   1:  PR[91,2] = PR[90,2] + -2.008;
   1:  PR[91,3] = PR[90,3] + 3.667;
   1:L PR[91] R[100]mm/sec CNT100;
   1:  PR[91,1] = PR[90,1] + -36.732;
   1:  PR[91,2] = PR[90,2] + -2.668;
   1:  PR[91,3] = PR[90,3] + 3.670;
   1:L PR[91] R[100]mm/sec CNT100;
   1:  PR[91,1] = PR[90,1] + -36.503;
   1:  PR[91,2] = PR[90,2] + -3.709;
   1:  PR[91,3] = PR[90,3] + 3.674;
   1:L PR[91] R[100]mm/sec CNT100;
   1:  PR[91,1] = PR[90,1] + -36.318;
   1:  PR[91,2] = PR[90,2] + -4.391;
   1:  PR[91,3] = PR[90,3] + 3.681;
   1:L PR[91] R[100]mm/sec CNT100;
   1:  PR[91,1] = PR[90,1] + -35.924;
   1:  PR[91,2] = PR[90,2] + -5.558;
   1:  PR[91,3] = PR[90,3] + 3.685;
   1:L PR[91] R[100]mm/sec CNT100;
   1:  PR[91,1] = PR[90,1] + -35.717;
   1:  PR[91,2] = PR[90,2] + -6.077;
   1:  PR[91,3] = PR[90,3] + 3.693;
   1:L PR[91] R[100]mm/sec CNT100;
   1:  PR[91,1] = PR[90,1] + -35.452;
   1:  PR[91,2] = PR[90,2] + -6.678;
   1:  PR[91,3] = PR[90,3] + 3.696;
   1:L PR[91] R[100]mm/sec CNT100;
   1:  PR[91,1] = PR[90,1] + -35.136;
   1:  PR[91,2] = PR[90,2] + -7.322;
   1:  PR[91,3] = PR[90,3] + 3.700;
   1:L PR[91] R[100]mm/sec CNT100;
   1:  PR[91,1] = PR[90,1] + -34.899;
   1:  PR[91,2] = PR[90,2] + -7.767;
   1:  PR[91,3] = PR[90,3] + 3.704;
   1:L PR[91] R[100]mm/sec CNT100;
   1:  PR[91,1] = PR[90,1] + -34.544;
   1:  PR[91,2] = PR[90,2] + -8.374;
   1:  PR[91,3] = PR[90,3] + 3.708;
   1:L PR[91] R[100]mm/sec CNT100;
   1:  PR[91,1] = PR[90,1] + -33.978;
   1:  PR[91,2] = PR[90,2] + -9.242;
   1:  PR[91,3] = PR[90,3] + 3.712;
   1:L PR[91] R[100]mm/sec CNT100;
   1:  PR[91,1] = PR[90,1] + -33.867;
   1:  PR[91,2] = PR[90,2] + -9.398;
   1:  PR[91,3] = PR[90,3] + 3.718;
   1:L PR[91] R[100]mm/sec CNT100;
   1:  PR[91,1] = PR[90,1] + -33.245;
   1:  PR[91,2] = PR[90,2] + -10.215;
   1:  PR[91,3] = PR[90,3] + 3.719;
   1:L PR[91] R[100]mm/sec CNT100;
   1:  PR[91,1] = PR[90,1] + -32.790;
   1:  PR[91,2] = PR[90,2] + -10.756;
   1:  PR[91,3] = PR[90,3] + 3.725;
   1:L PR[91] R[100]mm/sec CNT100;
   1:  PR[91,1] = PR[90,1] + -31.941;
   1:  PR[91,2] = PR[90,2] + -11.649;
   1:  PR[91,3] = PR[90,3] + 3.730;
   1:L PR[91] R[100]mm/sec CNT100;
   1:  PR[91,1] = PR[90,1] + -31.042;
   1:  PR[91,2] = PR[90,2] + -12.468;
   1:  PR[91,3] = PR[90,3] + 3.737;
   1:L PR[91] R[100]mm/sec CNT100;
   1:  PR[91,1] = PR[90,1] + -30.081;
   1:  PR[91,2] = PR[90,2] + -13.224;
   1:  PR[91,3] = PR[90,3] + 3.745;
   1:L PR[91] R[100]mm/sec CNT100;
   1:  PR[91,1] = PR[90,1] + -29.069;
   1:  PR[91,2] = PR[90,2] + -13.908;
   1:  PR[91,3] = PR[90,3] + 3.752;
   1:L PR[91] R[100]mm/sec CNT100;
   1:  PR[91,1] = PR[90,1] + -27.991;
   1:  PR[91,2] = PR[90,2] + -14.526;
   1:  PR[91,3] = PR[90,3] + 3.759;
   1:L PR[91] R[100]mm/sec CNT100;
   1:  PR[91,1] = PR[90,1] + -26.909;
   1:  PR[91,2] = PR[90,2] + -15.048;
   1:  PR[91,3] = PR[90,3] + 3.767;
   1:L PR[91] R[100]mm/sec CNT100;
   1:  PR[91,1] = PR[90,1] + -25.772;
   1:  PR[91,2] = PR[90,2] + -15.498;
   1:  PR[91,3] = PR[90,3] + 3.774;
   1:L PR[91] R[100]mm/sec CNT100;
   1:  PR[91,1] = PR[90,1] + -24.607;
   1:  PR[91,2] = PR[90,2] + -15.865;
   1:  PR[91,3] = PR[90,3] + 3.782;
   1:L PR[91] R[100]mm/sec CNT100;
   1:  PR[91,1] = PR[90,1] + -23.417;
   1:  PR[91,2] = PR[90,2] + -16.147;
   1:  PR[91,3] = PR[90,3] + 3.789;
   1:L PR[91] R[100]mm/sec CNT100;
   1:  PR[91,1] = PR[90,1] + -22.211;
   1:  PR[91,2] = PR[90,2] + -16.342;
   1:  PR[91,3] = PR[90,3] + 3.797;
   1:L PR[91] R[100]mm/sec CNT100;
   1:  PR[91,1] = PR[90,1] + -20.993;
   1:  PR[91,2] = PR[90,2] + -16.449;
   1:  PR[91,3] = PR[90,3] + 3.804;
   1:L PR[91] R[100]mm/sec CNT100;
   1:  PR[91,1] = PR[90,1] + -19.771;
   1:  PR[91,2] = PR[90,2] + -16.468;
   1:  PR[91,3] = PR[90,3] + 3.811;
   1:L PR[91] R[100]mm/sec CNT100;
   1:  PR[91,1] = PR[90,1] + -18.551;
   1:  PR[91,2] = PR[90,2] + -16.399;
   1:  PR[91,3] = PR[90,3] + 3.819;
   1:L PR[91] R[100]mm/sec CNT100;
   1:  PR[91,1] = PR[90,1] + -17.336;
   1:  PR[91,2] = PR[90,2] + -16.241;
   1:  PR[91,3] = PR[90,3] + 3.826;
   1:L PR[91] R[100]mm/sec CNT100;
   1:  PR[91,1] = PR[90,1] + -16.641;
   1:  PR[91,2] = PR[90,2] + -16.109;
   1:  PR[91,3] = PR[90,3] + 3.834;
   1:L PR[91] R[100]mm/sec CNT100;
   1:  PR[91,1] = PR[90,1] + -15.647;
   1:  PR[91,2] = PR[90,2] + -15.868;
   1:  PR[91,3] = PR[90,3] + 3.838;
   1:L PR[91] R[100]mm/sec CNT100;
   1:  PR[91,1] = PR[90,1] + -14.969;
   1:  PR[91,2] = PR[90,2] + -15.668;
   1:  PR[91,3] = PR[90,3] + 3.844;
   1:L PR[91] R[100]mm/sec CNT100;
   1:  PR[91,1] = PR[90,1] + -13.816;
   1:  PR[91,2] = PR[90,2] + -15.252;
   1:  PR[91,3] = PR[90,3] + 3.849;
   1:L PR[91] R[100]mm/sec CNT100;
   1:  PR[91,1] = PR[90,1] + -12.694;
   1:  PR[91,2] = PR[90,2] + -14.753;
   1:  PR[91,3] = PR[90,3] + 3.856;
   1:L PR[91] R[100]mm/sec CNT100;
   1:  PR[91,1] = PR[90,1] + -12.188;
   1:  PR[91,2] = PR[90,2] + -14.495;
   1:  PR[91,3] = PR[90,3] + 3.863;
   1:L PR[91] R[100]mm/sec CNT100;
   1:  PR[91,1] = PR[90,1] + -11.625;
   1:  PR[91,2] = PR[90,2] + -14.182;
   1:  PR[91,3] = PR[90,3] + 3.867;
   1:L PR[91] R[100]mm/sec CNT100;
   1:  PR[91,1] = PR[90,1] + -10.584;
   1:  PR[91,2] = PR[90,2] + -13.525;
   1:  PR[91,3] = PR[90,3] + 3.871;
   1:L PR[91] R[100]mm/sec CNT100;
   1:  PR[91,1] = PR[90,1] + -10.006;
   1:  PR[91,2] = PR[90,2] + -13.110;
   1:  PR[91,3] = PR[90,3] + 3.878;
   1:L PR[91] R[100]mm/sec CNT100;
   1:  PR[91,1] = PR[90,1] + -9.605;
   1:  PR[91,2] = PR[90,2] + -12.803;
   1:  PR[91,3] = PR[90,3] + 3.883;
   1:L PR[91] R[100]mm/sec CNT100;
   1:  PR[91,1] = PR[90,1] + -9.053;
   1:  PR[91,2] = PR[90,2] + -12.343;
   1:  PR[91,3] = PR[90,3] + 3.886;
   1:L PR[91] R[100]mm/sec CNT100;
   1:  PR[91,1] = PR[90,1] + -8.675;
   1:  PR[91,2] = PR[90,2] + -12.008;
   1:  PR[91,3] = PR[90,3] + 3.890;
   1:L PR[91] R[100]mm/sec CNT100;
   1:  PR[91,1] = PR[90,1] + -8.249;
   1:  PR[91,2] = PR[90,2] + -11.602;
   1:  PR[91,3] = PR[90,3] + 3.893;
   1:L PR[91] R[100]mm/sec CNT100;
   1:  PR[91,1] = PR[90,1] + -7.807;
   1:  PR[91,2] = PR[90,2] + -11.149;
   1:  PR[91,3] = PR[90,3] + 3.897;
   1:L PR[91] R[100]mm/sec CNT100;
   1:  PR[91,1] = PR[90,1] + -7.328;
   1:  PR[91,2] = PR[90,2] + -10.615;
   1:  PR[91,3] = PR[90,3] + 3.901;
   1:L PR[91] R[100]mm/sec CNT100;
   1:  PR[91,1] = PR[90,1] + -7.003;
   1:  PR[91,2] = PR[90,2] + -10.229;
   1:  PR[91,3] = PR[90,3] + 3.905;
   1:L PR[91] R[100]mm/sec CNT100;
   1:  PR[91,1] = PR[90,1] + -6.563;
   1:  PR[91,2] = PR[90,2] + -9.662;
   1:  PR[91,3] = PR[90,3] + 3.908;
   1:L PR[91] R[100]mm/sec CNT100;
   1:  PR[91,1] = PR[90,1] + -6.266;
   1:  PR[91,2] = PR[90,2] + -9.252;
   1:  PR[91,3] = PR[90,3] + 3.912;
   1:L PR[91] R[100]mm/sec CNT100;
   1:  PR[91,1] = PR[90,1] + -5.929;
   1:  PR[91,2] = PR[90,2] + -8.750;
   1:  PR[91,3] = PR[90,3] + 3.915;
   1:L PR[91] R[100]mm/sec CNT100;
   1:  PR[91,1] = PR[90,1] + -5.606;
   1:  PR[91,2] = PR[90,2] + -8.230;
   1:  PR[91,3] = PR[90,3] + 3.919;
   1:L PR[91] R[100]mm/sec CNT100;
   1:  PR[91,1] = PR[90,1] + -5.014;
   1:  PR[91,2] = PR[90,2] + -7.151;
   1:  PR[91,3] = PR[90,3] + 3.923;
   1:L PR[91] R[100]mm/sec CNT100;
   1:  PR[91,1] = PR[90,1] + -4.709;
   1:  PR[91,2] = PR[90,2] + -6.506;
   1:  PR[91,3] = PR[90,3] + 3.930;
   1:L PR[91] R[100]mm/sec CNT100;
   1:  PR[91,1] = PR[90,1] + -4.497;
   1:  PR[91,2] = PR[90,2] + -6.019;
   1:  PR[91,3] = PR[90,3] + 3.935;
   1:L PR[91] R[100]mm/sec CNT100;
   1:  PR[91,1] = PR[90,1] + -4.081;
   1:  PR[91,2] = PR[90,2] + -4.898;
   1:  PR[91,3] = PR[90,3] + 3.938;
   1:L PR[91] R[100]mm/sec CNT100;
   1:  PR[91,1] = PR[90,1] + -3.737;
   1:  PR[91,2] = PR[90,2] + -3.724;
   1:  PR[91,3] = PR[90,3] + 3.945;
   1:L PR[91] R[100]mm/sec CNT100;
   1:  PR[91,1] = PR[90,1] + -3.411;
   1:  PR[91,2] = PR[90,2] + -2.233;
   1:  PR[91,3] = PR[90,3] + 3.952;
   1:L PR[91] R[100]mm/sec CNT100;
   1:  PR[91,1] = PR[90,1] + -3.339;
   1:  PR[91,2] = PR[90,2] + -2.005;
   1:  PR[91,3] = PR[90,3] + 3.962;
   1:L PR[91] R[100]mm/sec CNT100;
   1:  PR[91,1] = PR[90,1] + -3.218;
   1:  PR[91,2] = PR[90,2] + -1.723;
   1:  PR[91,3] = PR[90,3] + 3.963;
   1:L PR[91] R[100]mm/sec CNT100;
   1:  PR[91,1] = PR[90,1] + -3.110;
   1:  PR[91,2] = PR[90,2] + -1.517;
   1:  PR[91,3] = PR[90,3] + 3.965;
   1:L PR[91] R[100]mm/sec CNT100;
   1:  PR[91,1] = PR[90,1] + -2.934;
   1:  PR[91,2] = PR[90,2] + -1.249;
   1:  PR[91,3] = PR[90,3] + 3.966;
   1:L PR[91] R[100]mm/sec CNT100;
   1:  PR[91,1] = PR[90,1] + -2.656;
   1:  PR[91,2] = PR[90,2] + -0.917;
   1:  PR[91,3] = PR[90,3] + 3.968;
   1:L PR[91] R[100]mm/sec CNT100;
   1:  PR[91,1] = PR[90,1] + -2.413;
   1:  PR[91,2] = PR[90,2] + -0.689;
   1:  PR[91,3] = PR[90,3] + 3.971;
   1:L PR[91] R[100]mm/sec CNT100;
   1:  PR[91,1] = PR[90,1] + -1.978;
   1:  PR[91,2] = PR[90,2] + -0.385;
   1:  PR[91,3] = PR[90,3] + 3.973;
   1:L PR[91] R[100]mm/sec CNT100;
   1:  PR[91,1] = PR[90,1] + -1.487;
   1:  PR[91,2] = PR[90,2] + -0.157;
   1:  PR[91,3] = PR[90,3] + 3.976;
   1:L PR[91] R[100]mm/sec CNT100;
   1:  PR[91,1] = PR[90,1] + -0.974;
   1:  PR[91,2] = PR[90,2] + -0.019;
   1:  PR[91,3] = PR[90,3] + 3.980;
   1:L PR[91] R[100]mm/sec CNT100;
   1:  PR[91,1] = PR[90,1] + -0.647;
   1:  PR[91,2] = PR[90,2] + 0.019;
   1:  PR[91,3] = PR[90,3] + 3.983;
   1:L PR[91] R[100]mm/sec CNT100;
   1:  PR[91,1] = PR[90,1] + 0.203;
   1:  PR[91,2] = PR[90,2] + 0.028;
   1:  PR[91,3] = PR[90,3] + 3.985;
   1:L PR[91] R[100]mm/sec CNT100;
   1:  PR[91] = PR[90];
   1:  PR[91,1] = PR[90,1] + 0.536;
   1:  PR[91,2] = PR[90,2] + 0.007;
   1:  PR[91,3] = PR[90,3] + 5.320;
   1:L PR[91] R[100]mm/sec CNT100;
   1:  PR[91,1] = PR[90,1] + 0.956;
   1:  PR[91,2] = PR[90,2] + -0.071;
   1:  PR[91,3] = PR[90,3] + 3.992;
   1:L PR[91] R[100]mm/sec CNT100;
   1:  PR[91,1] = PR[90,1] + 1.302;
   1:  PR[91,2] = PR[90,2] + -0.184;
   1:  PR[91,3] = PR[90,3] + 3.995;
   1:L PR[91] R[100]mm/sec CNT100;
   1:  PR[91,1] = PR[90,1] + 1.691;
   1:  PR[91,2] = PR[90,2] + -0.367;
   1:  PR[91,3] = PR[90,3] + 3.997;
   1:L PR[91] R[100]mm/sec CNT100;
   1:  PR[91,1] = PR[90,1] + 1.996;
   1:  PR[91,2] = PR[90,2] + -0.563;
   1:  PR[91,3] = PR[90,3] + 4.000;
   1:L PR[91] R[100]mm/sec CNT100;
   1:  PR[91,1] = PR[90,1] + 2.327;
   1:  PR[91,2] = PR[90,2] + -0.840;
   1:  PR[91,3] = PR[90,3] + 4.002;
   1:L PR[91] R[100]mm/sec CNT100;
   1:  PR[91,1] = PR[90,1] + 2.572;
   1:  PR[91,2] = PR[90,2] + -1.106;
   1:  PR[91,3] = PR[90,3] + 4.004;
   1:L PR[91] R[100]mm/sec CNT100;
   1:  PR[91,1] = PR[90,1] + 2.823;
   1:  PR[91,2] = PR[90,2] + -1.460;
   1:  PR[91,3] = PR[90,3] + 4.007;
   1:L PR[91] R[100]mm/sec CNT100;
   1:  PR[91,1] = PR[90,1] + 2.993;
   1:  PR[91,2] = PR[90,2] + -1.778;
   1:  PR[91,3] = PR[90,3] + 4.009;
   1:L PR[91] R[100]mm/sec CNT100;
   1:  PR[91,1] = PR[90,1] + 3.148;
   1:  PR[91,2] = PR[90,2] + -2.191;
   1:  PR[91,3] = PR[90,3] + 4.011;
   1:L PR[91] R[100]mm/sec CNT100;
   1:  PR[91,1] = PR[90,1] + 3.382;
   1:  PR[91,2] = PR[90,2] + -3.288;
   1:  PR[91,3] = PR[90,3] + 4.014;
   1:L PR[91] R[100]mm/sec CNT100;
   1:  PR[91,1] = PR[90,1] + 3.614;
   1:  PR[91,2] = PR[90,2] + -4.199;
   1:  PR[91,3] = PR[90,3] + 4.021;
   1:L PR[91] R[100]mm/sec CNT100;
   1:  PR[91,1] = PR[90,1] + 3.843;
   1:  PR[91,2] = PR[90,2] + -4.939;
   1:  PR[91,3] = PR[90,3] + 4.027;
   1:L PR[91] R[100]mm/sec CNT100;
   1:  PR[91,1] = PR[90,1] + 4.167;
   1:  PR[91,2] = PR[90,2] + -5.822;
   1:  PR[91,3] = PR[90,3] + 4.031;
   1:L PR[91] R[100]mm/sec CNT100;
   1:  PR[91,1] = PR[90,1] + 4.469;
   1:  PR[91,2] = PR[90,2] + -6.535;
   1:  PR[91,3] = PR[90,3] + 4.037;
   1:L PR[91] R[100]mm/sec CNT100;
   1:  PR[91,1] = PR[90,1] + 4.804;
   1:  PR[91,2] = PR[90,2] + -7.233;
   1:  PR[91,3] = PR[90,3] + 4.042;
   1:L PR[91] R[100]mm/sec CNT100;
   1:  PR[91,1] = PR[90,1] + 5.170;
   1:  PR[91,2] = PR[90,2] + -7.911;
   1:  PR[91,3] = PR[90,3] + 4.046;
   1:L PR[91] R[100]mm/sec CNT100;
   1:  PR[91,1] = PR[90,1] + 5.660;
   1:  PR[91,2] = PR[90,2] + -8.722;
   1:  PR[91,3] = PR[90,3] + 4.051;
   1:L PR[91] R[100]mm/sec CNT100;
   1:  PR[91,1] = PR[90,1] + 6.090;
   1:  PR[91,2] = PR[90,2] + -9.357;
   1:  PR[91,3] = PR[90,3] + 4.057;
   1:L PR[91] R[100]mm/sec CNT100;
   1:  PR[91,1] = PR[90,1] + 6.663;
   1:  PR[91,2] = PR[90,2] + -10.119;
   1:  PR[91,3] = PR[90,3] + 4.061;
   1:L PR[91] R[100]mm/sec CNT100;
   1:  PR[91,1] = PR[90,1] + 7.154;
   1:  PR[91,2] = PR[90,2] + -10.705;
   1:  PR[91,3] = PR[90,3] + 4.067;
   1:L PR[91] R[100]mm/sec CNT100;
   1:  PR[91,1] = PR[90,1] + 7.807;
   1:  PR[91,2] = PR[90,2] + -11.409;
   1:  PR[91,3] = PR[90,3] + 4.072;
   1:L PR[91] R[100]mm/sec CNT100;
   1:  PR[91,1] = PR[90,1] + 8.355;
   1:  PR[91,2] = PR[90,2] + -11.943;
   1:  PR[91,3] = PR[90,3] + 4.078;
   1:L PR[91] R[100]mm/sec CNT100;
   1:  PR[91,1] = PR[90,1] + 8.924;
   1:  PR[91,2] = PR[90,2] + -12.450;
   1:  PR[91,3] = PR[90,3] + 4.082;
   1:L PR[91] R[100]mm/sec CNT100;
   1:  PR[91,1] = PR[90,1] + 9.514;
   1:  PR[91,2] = PR[90,2] + -12.928;
   1:  PR[91,3] = PR[90,3] + 4.087;
   1:L PR[91] R[100]mm/sec CNT100;
   1:  PR[91,1] = PR[90,1] + 10.121;
   1:  PR[91,2] = PR[90,2] + -13.376;
   1:  PR[91,3] = PR[90,3] + 4.092;
   1:L PR[91] R[100]mm/sec CNT100;
   1:  PR[91,1] = PR[90,1] + 10.930;
   1:  PR[91,2] = PR[90,2] + -13.915;
   1:  PR[91,3] = PR[90,3] + 4.096;
   1:L PR[91] R[100]mm/sec CNT100;
   1:  PR[91,1] = PR[90,1] + 11.575;
   1:  PR[91,2] = PR[90,2] + -14.296;
   1:  PR[91,3] = PR[90,3] + 4.102;
   1:L PR[91] R[100]mm/sec CNT100;
   1:  PR[91,1] = PR[90,1] + 12.441;
   1:  PR[91,2] = PR[90,2] + -14.753;
   1:  PR[91,3] = PR[90,3] + 4.107;
   1:L PR[91] R[100]mm/sec CNT100;
   1:  PR[91,1] = PR[90,1] + 13.119;
   1:  PR[91,2] = PR[90,2] + -15.066;
   1:  PR[91,3] = PR[90,3] + 4.113;
   1:L PR[91] R[100]mm/sec CNT100;
   1:  PR[91,1] = PR[90,1] + 14.035;
   1:  PR[91,2] = PR[90,2] + -15.434;
   1:  PR[91,3] = PR[90,3] + 4.117;
   1:L PR[91] R[100]mm/sec CNT100;
   1:  PR[91,1] = PR[90,1] + 14.741;
   1:  PR[91,2] = PR[90,2] + -15.676;
   1:  PR[91,3] = PR[90,3] + 4.123;
   1:L PR[91] R[100]mm/sec CNT100;
   1:  PR[91,1] = PR[90,1] + 15.454;
   1:  PR[91,2] = PR[90,2] + -15.886;
   1:  PR[91,3] = PR[90,3] + 4.128;
   1:L PR[91] R[100]mm/sec CNT100;
   1:  PR[91,1] = PR[90,1] + 16.423;
   1:  PR[91,2] = PR[90,2] + -16.118;
   1:  PR[91,3] = PR[90,3] + 4.132;
   1:L PR[91] R[100]mm/sec CNT100;
   1:  PR[91,1] = PR[90,1] + 17.149;
   1:  PR[91,2] = PR[90,2] + -16.253;
   1:  PR[91,3] = PR[90,3] + 4.138;
   1:L PR[91] R[100]mm/sec CNT100;
   1:  PR[91,1] = PR[90,1] + 18.143;
   1:  PR[91,2] = PR[90,2] + -16.384;
   1:  PR[91,3] = PR[90,3] + 4.143;
   1:L PR[91] R[100]mm/sec CNT100;
   1:  PR[91,1] = PR[90,1] + 18.879;
   1:  PR[91,2] = PR[90,2] + -16.444;
   1:  PR[91,3] = PR[90,3] + 4.149;
   1:L PR[91] R[100]mm/sec CNT100;
   1:  PR[91,1] = PR[90,1] + 19.615;
   1:  PR[91,2] = PR[90,2] + -16.471;
   1:  PR[91,3] = PR[90,3] + 4.153;
   1:L PR[91] R[100]mm/sec CNT100;
   1:  PR[91,1] = PR[90,1] + 20.625;
   1:  PR[91,2] = PR[90,2] + -16.456;
   1:  PR[91,3] = PR[90,3] + 4.158;
   1:L PR[91] R[100]mm/sec CNT100;
   1:  PR[91,1] = PR[90,1] + 21.357;
   1:  PR[91,2] = PR[90,2] + -16.408;
   1:  PR[91,3] = PR[90,3] + 4.164;
   1:L PR[91] R[100]mm/sec CNT100;
   1:  PR[91,1] = PR[90,1] + 22.083;
   1:  PR[91,2] = PR[90,2] + -16.328;
   1:  PR[91,3] = PR[90,3] + 4.168;
   1:L PR[91] R[100]mm/sec CNT100;
   1:  PR[91,1] = PR[90,1] + 23.089;
   1:  PR[91,2] = PR[90,2] + -16.165;
   1:  PR[91,3] = PR[90,3] + 4.173;
   1:L PR[91] R[100]mm/sec CNT100;
   1:  PR[91,1] = PR[90,1] + 23.801;
   1:  PR[91,2] = PR[90,2] + -16.011;
   1:  PR[91,3] = PR[90,3] + 4.179;
   1:L PR[91] R[100]mm/sec CNT100;
   1:  PR[91,1] = PR[90,1] + 24.503;
   1:  PR[91,2] = PR[90,2] + -15.826;
   1:  PR[91,3] = PR[90,3] + 4.183;
   1:L PR[91] R[100]mm/sec CNT100;
   1:  PR[91,1] = PR[90,1] + 25.480;
   1:  PR[91,2] = PR[90,2] + -15.516;
   1:  PR[91,3] = PR[90,3] + 4.188;
   1:L PR[91] R[100]mm/sec CNT100;
   1:  PR[91,1] = PR[90,1] + 26.155;
   1:  PR[91,2] = PR[90,2] + -15.262;
   1:  PR[91,3] = PR[90,3] + 4.194;
   1:L PR[91] R[100]mm/sec CNT100;
   1:  PR[91,1] = PR[90,1] + 27.100;
   1:  PR[91,2] = PR[90,2] + -14.850;
   1:  PR[91,3] = PR[90,3] + 4.198;
   1:L PR[91] R[100]mm/sec CNT100;
   1:  PR[91,1] = PR[90,1] + 27.747;
   1:  PR[91,2] = PR[90,2] + -14.527;
   1:  PR[91,3] = PR[90,3] + 4.205;
   1:L PR[91] R[100]mm/sec CNT100;
   1:  PR[91,1] = PR[90,1] + 28.376;
   1:  PR[91,2] = PR[90,2] + -14.178;
   1:  PR[91,3] = PR[90,3] + 4.209;
   1:L PR[91] R[100]mm/sec CNT100;
   1:  PR[91,1] = PR[90,1] + 29.256;
   1:  PR[91,2] = PR[90,2] + -13.630;
   1:  PR[91,3] = PR[90,3] + 4.213;
   1:L PR[91] R[100]mm/sec CNT100;
   1:  PR[91,1] = PR[90,1] + 29.845;
   1:  PR[91,2] = PR[90,2] + -13.219;
   1:  PR[91,3] = PR[90,3] + 4.220;
   1:L PR[91] R[100]mm/sec CNT100;
   1:  PR[91,1] = PR[90,1] + 30.415;
   1:  PR[91,2] = PR[90,2] + -12.783;
   1:  PR[91,3] = PR[90,3] + 4.224;
   1:L PR[91] R[100]mm/sec CNT100;
   1:  PR[91,1] = PR[90,1] + 31.208;
   1:  PR[91,2] = PR[90,2] + -12.109;
   1:  PR[91,3] = PR[90,3] + 4.228;
   1:L PR[91] R[100]mm/sec CNT100;
   1:  PR[91,1] = PR[90,1] + 31.729;
   1:  PR[91,2] = PR[90,2] + -11.618;
   1:  PR[91,3] = PR[90,3] + 4.235;
   1:L PR[91] R[100]mm/sec CNT100;
   1:  PR[91,1] = PR[90,1] + 32.227;
   1:  PR[91,2] = PR[90,2] + -11.106;
   1:  PR[91,3] = PR[90,3] + 4.239;
   1:L PR[91] R[100]mm/sec CNT100;
   1:  PR[91,1] = PR[90,1] + 32.917;
   1:  PR[91,2] = PR[90,2] + -10.321;
   1:  PR[91,3] = PR[90,3] + 4.244;
   1:L PR[91] R[100]mm/sec CNT100;
   1:  PR[91,1] = PR[90,1] + 33.357;
   1:  PR[91,2] = PR[90,2] + -9.763;
   1:  PR[91,3] = PR[90,3] + 4.250;
   1:L PR[91] R[100]mm/sec CNT100;
   1:  PR[91,1] = PR[90,1] + 33.962;
   1:  PR[91,2] = PR[90,2] + -8.908;
   1:  PR[91,3] = PR[90,3] + 4.254;
   1:L PR[91] R[100]mm/sec CNT100;
   1:  PR[91,1] = PR[90,1] + 34.344;
   1:  PR[91,2] = PR[90,2] + -8.306;
   1:  PR[91,3] = PR[90,3] + 4.261;
   1:L PR[91] R[100]mm/sec CNT100;
   1:  PR[91,1] = PR[90,1] + 34.698;
   1:  PR[91,2] = PR[90,2] + -7.689;
   1:  PR[91,3] = PR[90,3] + 4.265;
   1:L PR[91] R[100]mm/sec CNT100;
   1:  PR[91,1] = PR[90,1] + 35.174;
   1:  PR[91,2] = PR[90,2] + -6.752;
   1:  PR[91,3] = PR[90,3] + 4.269;
   1:L PR[91] R[100]mm/sec CNT100;
   1:  PR[91,1] = PR[90,1] + 35.462;
   1:  PR[91,2] = PR[90,2] + -6.103;
   1:  PR[91,3] = PR[90,3] + 4.276;
   1:L PR[91] R[100]mm/sec CNT100;
   1:  PR[91,1] = PR[90,1] + 35.722;
   1:  PR[91,2] = PR[90,2] + -5.442;
   1:  PR[91,3] = PR[90,3] + 4.280;
   1:L PR[91] R[100]mm/sec CNT100;
   1:  PR[91,1] = PR[90,1] + 36.058;
   1:  PR[91,2] = PR[90,2] + -4.445;
   1:  PR[91,3] = PR[90,3] + 4.284;
   1:L PR[91] R[100]mm/sec CNT100;
   1:  PR[91,1] = PR[90,1] + 36.247;
   1:  PR[91,2] = PR[90,2] + -3.764;
   1:  PR[91,3] = PR[90,3] + 4.291;
   1:L PR[91] R[100]mm/sec CNT100;
   1:  PR[91,1] = PR[90,1] + 36.476;
   1:  PR[91,2] = PR[90,2] + -2.736;
   1:  PR[91,3] = PR[90,3] + 4.295;
   1:L PR[91] R[100]mm/sec CNT100;
   1:  PR[91,1] = PR[90,1] + 36.595;
   1:  PR[91,2] = PR[90,2] + -2.036;
   1:  PR[91,3] = PR[90,3] + 4.301;
   1:L PR[91] R[100]mm/sec CNT100;
   1:  PR[91,1] = PR[90,1] + 36.683;
   1:  PR[91,2] = PR[90,2] + -1.333;
   1:  PR[91,3] = PR[90,3] + 4.306;
   1:L PR[91] R[100]mm/sec CNT100;
   1:  PR[91,1] = PR[90,1] + 36.760;
   1:  PR[91,2] = PR[90,2] + -0.281;
   1:  PR[91,3] = PR[90,3] + 4.310;
   1:L PR[91] R[100]mm/sec CNT100;
   1:  PR[91,1] = PR[90,1] + 36.775;
   1:  PR[91,2] = PR[90,2] + 0.428;
   1:  PR[91,3] = PR[90,3] + 4.316;
   1:L PR[91] R[100]mm/sec CNT100;
   1:  PR[91,1] = PR[90,1] + 36.760;
   1:  PR[91,2] = PR[90,2] + 1.137;
   1:  PR[91,3] = PR[90,3] + 4.321;
   1:L PR[91] R[100]mm/sec CNT100;
   1:  PR[91,1] = PR[90,1] + 36.683;
   1:  PR[91,2] = PR[90,2] + 2.188;
   1:  PR[91,3] = PR[90,3] + 4.325;
   1:L PR[91] R[100]mm/sec CNT100;
   1:  PR[91,1] = PR[90,1] + 36.595;
   1:  PR[91,2] = PR[90,2] + 2.892;
   1:  PR[91,3] = PR[90,3] + 4.331;
   1:L PR[91] R[100]mm/sec CNT100;
   1:  PR[91,1] = PR[90,1] + 36.476;
   1:  PR[91,2] = PR[90,2] + 3.591;
   1:  PR[91,3] = PR[90,3] + 4.336;
   1:L PR[91] R[100]mm/sec CNT100;
   1:  PR[91,1] = PR[90,1] + 36.247;
   1:  PR[91,2] = PR[90,2] + 4.619;
   1:  PR[91,3] = PR[90,3] + 4.340;
   1:L PR[91] R[100]mm/sec CNT100;
   1:  PR[91,1] = PR[90,1] + 36.058;
   1:  PR[91,2] = PR[90,2] + 5.300;
   1:  PR[91,3] = PR[90,3] + 4.346;
   1:L PR[91] R[100]mm/sec CNT100;
   1:  PR[91,1] = PR[90,1] + 35.722;
   1:  PR[91,2] = PR[90,2] + 6.297;
   1:  PR[91,3] = PR[90,3] + 4.351;
   1:L PR[91] R[100]mm/sec CNT100;
   1:  PR[91,1] = PR[90,1] + 35.462;
   1:  PR[91,2] = PR[90,2] + 6.958;
   1:  PR[91,3] = PR[90,3] + 4.357;
   1:L PR[91] R[100]mm/sec CNT100;
   1:  PR[91,1] = PR[90,1] + 35.174;
   1:  PR[91,2] = PR[90,2] + 7.607;
   1:  PR[91,3] = PR[90,3] + 4.361;
   1:L PR[91] R[100]mm/sec CNT100;
   1:  PR[91,1] = PR[90,1] + 34.698;
   1:  PR[91,2] = PR[90,2] + 8.544;
   1:  PR[91,3] = PR[90,3] + 4.366;
   1:L PR[91] R[100]mm/sec CNT100;
   1:  PR[91,1] = PR[90,1] + 34.344;
   1:  PR[91,2] = PR[90,2] + 9.161;
   1:  PR[91,3] = PR[90,3] + 4.372;
   1:L PR[91] R[100]mm/sec CNT100;
   1:  PR[91,1] = PR[90,1] + 33.962;
   1:  PR[91,2] = PR[90,2] + 9.763;
   1:  PR[91,3] = PR[90,3] + 4.376;
   1:L PR[91] R[100]mm/sec CNT100;
   1:  PR[91,1] = PR[90,1] + 33.357;
   1:  PR[91,2] = PR[90,2] + 10.618;
   1:  PR[91,3] = PR[90,3] + 4.381;
   1:L PR[91] R[100]mm/sec CNT100;
   1:  PR[91,1] = PR[90,1] + 32.915;
   1:  PR[91,2] = PR[90,2] + 11.178;
   1:  PR[91,3] = PR[90,3] + 4.387;
   1:L PR[91] R[100]mm/sec CNT100;
   1:  PR[91,1] = PR[90,1] + 32.448;
   1:  PR[91,2] = PR[90,2] + 11.720;
   1:  PR[91,3] = PR[90,3] + 4.391;
   1:L PR[91] R[100]mm/sec CNT100;
   1:  PR[91,1] = PR[90,1] + 31.727;
   1:  PR[91,2] = PR[90,2] + 12.475;
   1:  PR[91,3] = PR[90,3] + 4.396;
   1:L PR[91] R[100]mm/sec CNT100;
   1:  PR[91,1] = PR[90,1] + 31.208;
   1:  PR[91,2] = PR[90,2] + 12.964;
   1:  PR[91,3] = PR[90,3] + 4.402;
   1:L PR[91] R[100]mm/sec CNT100;
   1:  PR[91,1] = PR[90,1] + 30.415;
   1:  PR[91,2] = PR[90,2] + 13.638;
   1:  PR[91,3] = PR[90,3] + 4.406;
   1:L PR[91] R[100]mm/sec CNT100;
   1:  PR[91,1] = PR[90,1] + 29.845;
   1:  PR[91,2] = PR[90,2] + 14.074;
   1:  PR[91,3] = PR[90,3] + 4.413;
   1:L PR[91] R[100]mm/sec CNT100;
   1:  PR[91,1] = PR[90,1] + 29.256;
   1:  PR[91,2] = PR[90,2] + 14.485;
   1:  PR[91,3] = PR[90,3] + 4.417;
   1:L PR[91] R[100]mm/sec CNT100;
   1:  PR[91,1] = PR[90,1] + 28.376;
   1:  PR[91,2] = PR[90,2] + 15.034;
   1:  PR[91,3] = PR[90,3] + 4.421;
   1:L PR[91] R[100]mm/sec CNT100;
   1:  PR[91,1] = PR[90,1] + 27.747;
   1:  PR[91,2] = PR[90,2] + 15.383;
   1:  PR[91,3] = PR[90,3] + 4.428;
   1:L PR[91] R[100]mm/sec CNT100;
   1:  PR[91,1] = PR[90,1] + 27.100;
   1:  PR[91,2] = PR[90,2] + 15.705;
   1:  PR[91,3] = PR[90,3] + 4.432;
   1:L PR[91] R[100]mm/sec CNT100;
   1:  PR[91,1] = PR[90,1] + 26.155;
   1:  PR[91,2] = PR[90,2] + 16.118;
   1:  PR[91,3] = PR[90,3] + 4.437;
   1:L PR[91] R[100]mm/sec CNT100;
   1:  PR[91,1] = PR[90,1] + 25.478;
   1:  PR[91,2] = PR[90,2] + 16.372;
   1:  PR[91,3] = PR[90,3] + 4.443;
   1:L PR[91] R[100]mm/sec CNT100;
   1:  PR[91,1] = PR[90,1] + 24.787;
   1:  PR[91,2] = PR[90,2] + 16.598;
   1:  PR[91,3] = PR[90,3] + 4.447;
   1:L PR[91] R[100]mm/sec CNT100;
   1:  PR[91,1] = PR[90,1] + 23.798;
   1:  PR[91,2] = PR[90,2] + 16.866;
   1:  PR[91,3] = PR[90,3] + 4.452;
   1:L PR[91] R[100]mm/sec CNT100;
   1:  PR[91,1] = PR[90,1] + 23.089;
   1:  PR[91,2] = PR[90,2] + 17.020;
   1:  PR[91,3] = PR[90,3] + 4.458;
   1:L PR[91] R[100]mm/sec CNT100;
   1:  PR[91,1] = PR[90,1] + 22.083;
   1:  PR[91,2] = PR[90,2] + 17.183;
   1:  PR[91,3] = PR[90,3] + 4.462;
   1:L PR[91] R[100]mm/sec CNT100;
   1:  PR[91,1] = PR[90,1] + 21.357;
   1:  PR[91,2] = PR[90,2] + 17.263;
   1:  PR[91,3] = PR[90,3] + 4.468;
   1:L PR[91] R[100]mm/sec CNT100;
   1:  PR[91,1] = PR[90,1] + 20.625;
   1:  PR[91,2] = PR[90,2] + 17.312;
   1:  PR[91,3] = PR[90,3] + 4.473;
   1:L PR[91] R[100]mm/sec CNT100;
   1:  PR[91,1] = PR[90,1] + 19.615;
   1:  PR[91,2] = PR[90,2] + 17.327;
   1:  PR[91,3] = PR[90,3] + 4.477;
   1:L PR[91] R[100]mm/sec CNT100;
   1:  PR[91,1] = PR[90,1] + 18.882;
   1:  PR[91,2] = PR[90,2] + 17.300;
   1:  PR[91,3] = PR[90,3] + 4.483;
   1:L PR[91] R[100]mm/sec CNT100;
   1:  PR[91,1] = PR[90,1] + 17.882;
   1:  PR[91,2] = PR[90,2] + 17.210;
   1:  PR[91,3] = PR[90,3] + 4.488;
   1:L PR[91] R[100]mm/sec CNT100;
   1:  PR[91,1] = PR[90,1] + 17.151;
   1:  PR[91,2] = PR[90,2] + 17.108;
   1:  PR[91,3] = PR[90,3] + 4.494;
   1:L PR[91] R[100]mm/sec CNT100;
   1:  PR[91,1] = PR[90,1] + 16.421;
   1:  PR[91,2] = PR[90,2] + 16.973;
   1:  PR[91,3] = PR[90,3] + 4.498;
   1:L PR[91] R[100]mm/sec CNT100;
   1:  PR[91,1] = PR[90,1] + 15.694;
   1:  PR[91,2] = PR[90,2] + 16.803;
   1:  PR[91,3] = PR[90,3] + 4.503;
   1:L PR[91] R[100]mm/sec CNT100;
   1:  PR[91,1] = PR[90,1] + 14.975;
   1:  PR[91,2] = PR[90,2] + 16.601;
   1:  PR[91,3] = PR[90,3] + 4.508;
   1:L PR[91] R[100]mm/sec CNT100;
   1:  PR[91,1] = PR[90,1] + 13.809;
   1:  PR[91,2] = PR[90,2] + 16.203;
   1:  PR[91,3] = PR[90,3] + 4.512;
   1:L PR[91] R[100]mm/sec CNT100;
   1:  PR[91,1] = PR[90,1] + 13.121;
   1:  PR[91,2] = PR[90,2] + 15.922;
   1:  PR[91,3] = PR[90,3] + 4.520;
   1:L PR[91] R[100]mm/sec CNT100;
   1:  PR[91,1] = PR[90,1] + 12.441;
   1:  PR[91,2] = PR[90,2] + 15.608;
   1:  PR[91,3] = PR[90,3] + 4.524;
   1:L PR[91] R[100]mm/sec CNT100;
   1:  PR[91,1] = PR[90,1] + 11.575;
   1:  PR[91,2] = PR[90,2] + 15.151;
   1:  PR[91,3] = PR[90,3] + 4.529;
   1:L PR[91] R[100]mm/sec CNT100;
   1:  PR[91,1] = PR[90,1] + 10.928;
   1:  PR[91,2] = PR[90,2] + 14.769;
   1:  PR[91,3] = PR[90,3] + 4.535;
   1:L PR[91] R[100]mm/sec CNT100;
   1:  PR[91,1] = PR[90,1] + 10.295;
   1:  PR[91,2] = PR[90,2] + 14.354;
   1:  PR[91,3] = PR[90,3] + 4.539;
   1:L PR[91] R[100]mm/sec CNT100;
   1:  PR[91,1] = PR[90,1] + 9.678;
   1:  PR[91,2] = PR[90,2] + 13.909;
   1:  PR[91,3] = PR[90,3] + 4.544;
   1:L PR[91] R[100]mm/sec CNT100;
   1:  PR[91,1] = PR[90,1] + 9.083;
   1:  PR[91,2] = PR[90,2] + 13.435;
   1:  PR[91,3] = PR[90,3] + 4.548;
   1:L PR[91] R[100]mm/sec CNT100;
   1:  PR[91,1] = PR[90,1] + 8.210;
   1:  PR[91,2] = PR[90,2] + 12.660;
   1:  PR[91,3] = PR[90,3] + 4.553;
   1:L PR[91] R[100]mm/sec CNT100;
   1:  PR[91,1] = PR[90,1] + 7.672;
   1:  PR[91,2] = PR[90,2] + 12.126;
   1:  PR[91,3] = PR[90,3] + 4.560;
   1:L PR[91] R[100]mm/sec CNT100;
   1:  PR[91,1] = PR[90,1] + 7.155;
   1:  PR[91,2] = PR[90,2] + 11.562;
   1:  PR[91,3] = PR[90,3] + 4.565;
   1:L PR[91] R[100]mm/sec CNT100;
   1:  PR[91,1] = PR[90,1] + 6.664;
   1:  PR[91,2] = PR[90,2] + 10.974;
   1:  PR[91,3] = PR[90,3] + 4.569;
   1:L PR[91] R[100]mm/sec CNT100;
   1:  PR[91,1] = PR[90,1] + 6.090;
   1:  PR[91,2] = PR[90,2] + 10.213;
   1:  PR[91,3] = PR[90,3] + 4.574;
   1:L PR[91] R[100]mm/sec CNT100;
   1:  PR[91,1] = PR[90,1] + 5.660;
   1:  PR[91,2] = PR[90,2] + 9.577;
   1:  PR[91,3] = PR[90,3] + 4.580;
   1:L PR[91] R[100]mm/sec CNT100;
   1:  PR[91,1] = PR[90,1] + 5.170;
   1:  PR[91,2] = PR[90,2] + 8.767;
   1:  PR[91,3] = PR[90,3] + 4.584;
   1:L PR[91] R[100]mm/sec CNT100;
   1:  PR[91,1] = PR[90,1] + 4.804;
   1:  PR[91,2] = PR[90,2] + 8.088;
   1:  PR[91,3] = PR[90,3] + 4.590;
   1:L PR[91] R[100]mm/sec CNT100;
   1:  PR[91,1] = PR[90,1] + 4.470;
   1:  PR[91,2] = PR[90,2] + 7.392;
   1:  PR[91,3] = PR[90,3] + 4.595;
   1:L PR[91] R[100]mm/sec CNT100;
   1:  PR[91,1] = PR[90,1] + 4.106;
   1:  PR[91,2] = PR[90,2] + 6.523;
   1:  PR[91,3] = PR[90,3] + 4.600;
   1:L PR[91] R[100]mm/sec CNT100;
   1:  PR[91,1] = PR[90,1] + 3.843;
   1:  PR[91,2] = PR[90,2] + 5.795;
   1:  PR[91,3] = PR[90,3] + 4.605;
   1:L PR[91] R[100]mm/sec CNT100;
   1:  PR[91,1] = PR[90,1] + 3.614;
   1:  PR[91,2] = PR[90,2] + 5.053;
   1:  PR[91,3] = PR[90,3] + 4.610;
   1:L PR[91] R[100]mm/sec CNT100;
   1:  PR[91,1] = PR[90,1] + 3.419;
   1:  PR[91,2] = PR[90,2] + 4.300;
   1:  PR[91,3] = PR[90,3] + 4.615;
   1:L PR[91] R[100]mm/sec CNT100;
   1:  PR[91,1] = PR[90,1] + 3.222;
   1:  PR[91,2] = PR[90,2] + 3.354;
   1:  PR[91,3] = PR[90,3] + 4.619;
   1:L PR[91] R[100]mm/sec CNT100;
   1:  PR[91,1] = PR[90,1] + 3.119;
   1:  PR[91,2] = PR[90,2] + 2.958;
   1:  PR[91,3] = PR[90,3] + 4.625;
   1:L PR[91] R[100]mm/sec CNT100;
   1:  PR[91,1] = PR[90,1] + 2.991;
   1:  PR[91,2] = PR[90,2] + 2.629;
   1:  PR[91,3] = PR[90,3] + 4.628;
   1:L PR[91] R[100]mm/sec CNT100;
   1:  PR[91,1] = PR[90,1] + 2.823;
   1:  PR[91,2] = PR[90,2] + 2.315;
   1:  PR[91,3] = PR[90,3] + 4.630;
   1:L PR[91] R[100]mm/sec CNT100;
   1:  PR[91,1] = PR[90,1] + 2.569;
   1:  PR[91,2] = PR[90,2] + 1.957;
   1:  PR[91,3] = PR[90,3] + 4.632;
   1:L PR[91] R[100]mm/sec CNT100;
   1:  PR[91,1] = PR[90,1] + 2.268;
   1:  PR[91,2] = PR[90,2] + 1.642;
   1:  PR[91,3] = PR[90,3] + 4.635;
   1:L PR[91] R[100]mm/sec CNT100;
   1:  PR[91,1] = PR[90,1] + 1.993;
   1:  PR[91,2] = PR[90,2] + 1.416;
   1:  PR[91,3] = PR[90,3] + 4.637;
   1:L PR[91] R[100]mm/sec CNT100;
   1:  PR[91,1] = PR[90,1] + 1.691;
   1:  PR[91,2] = PR[90,2] + 1.222;
   1:  PR[91,3] = PR[90,3] + 4.640;
   1:L PR[91] R[100]mm/sec CNT100;
   1:  PR[91,1] = PR[90,1] + 1.302;
   1:  PR[91,2] = PR[90,2] + 1.039;
   1:  PR[91,3] = PR[90,3] + 4.642;
   1:L PR[91] R[100]mm/sec CNT100;
   1:  PR[91,1] = PR[90,1] + 0.956;
   1:  PR[91,2] = PR[90,2] + 0.926;
   1:  PR[91,3] = PR[90,3] + 4.644;
   1:L PR[91] R[100]mm/sec CNT100;
   1:  PR[91,1] = PR[90,1] + 0.536;
   1:  PR[91,2] = PR[90,2] + 0.848;
   1:  PR[91,3] = PR[90,3] + 4.647;
   1:L PR[91] R[100]mm/sec CNT100;
   1:  PR[91,1] = PR[90,1] + 0.191;
   1:  PR[91,2] = PR[90,2] + 0.828;
   1:  PR[91,3] = PR[90,3] + 4.649;
   1:L PR[91] R[100]mm/sec CNT100;
   1:  PR[91,1] = PR[90,1] + -0.431;
   1:  PR[91,3] = PR[90,3] + 4.651;
   1:L PR[91] R[100]mm/sec CNT100;
   1:  PR[91,1] = PR[90,1] + -0.775;
   1:  PR[91,2] = PR[90,2] + 0.848;
   1:  PR[91,3] = PR[90,3] + 4.655;
   1:L PR[91] R[100]mm/sec CNT100;
   1:  PR[91,1] = PR[90,1] + -1.194;
   1:  PR[91,2] = PR[90,2] + 0.926;
   1:  PR[91,3] = PR[90,3] + 4.657;
   1:L PR[91] R[100]mm/sec CNT100;
   1:  PR[91,1] = PR[90,1] + -1.538;
   1:  PR[91,2] = PR[90,2] + 1.038;
   1:  PR[91,3] = PR[90,3] + 4.660;
   1:L PR[91] R[100]mm/sec CNT100;
   1:  PR[91,1] = PR[90,1] + -1.866;
   1:  PR[91,2] = PR[90,2] + 1.189;
   1:  PR[91,3] = PR[90,3] + 4.662;
   1:L PR[91] R[100]mm/sec CNT100;
   1:  PR[91,1] = PR[90,1] + -2.293;
   1:  PR[91,2] = PR[90,2] + 1.462;
   1:  PR[91,3] = PR[90,3] + 4.664;
   1:L PR[91] R[100]mm/sec CNT100;
   1:  PR[91,1] = PR[90,1] + -2.568;
   1:  PR[91,2] = PR[90,2] + 1.698;
   1:  PR[91,3] = PR[90,3] + 4.667;
   1:L PR[91] R[100]mm/sec CNT100;
   1:  PR[91,1] = PR[90,1] + -2.811;
   1:  PR[91,2] = PR[90,2] + 1.961;
   1:  PR[91,3] = PR[90,3] + 4.669;
   1:L PR[91] R[100]mm/sec CNT100;
   1:  PR[91,1] = PR[90,1] + -3.062;
   1:  PR[91,2] = PR[90,2] + 2.315;
   1:  PR[91,3] = PR[90,3] + 4.672;
   1:L PR[91] R[100]mm/sec CNT100;
   1:  PR[91,1] = PR[90,1] + -3.231;
   1:  PR[91,2] = PR[90,2] + 2.633;
   1:  PR[91,3] = PR[90,3] + 4.674;
   1:L PR[91] R[100]mm/sec CNT100;
   1:  PR[91,1] = PR[90,1] + -3.387;
   1:  PR[91,2] = PR[90,2] + 3.047;
   1:  PR[91,3] = PR[90,3] + 4.676;
   1:L PR[91] R[100]mm/sec CNT100;
   1:  PR[91,1] = PR[90,1] + -3.620;
   1:  PR[91,2] = PR[90,2] + 4.143;
   1:  PR[91,3] = PR[90,3] + 4.679;
   1:L PR[91] R[100]mm/sec CNT100;
   1:  PR[91,1] = PR[90,1] + -3.852;
   1:  PR[91,2] = PR[90,2] + 5.054;
   1:  PR[91,3] = PR[90,3] + 4.686;
   1:L PR[91] R[100]mm/sec CNT100;
   1:  PR[91,1] = PR[90,1] + -4.081;
   1:  PR[91,2] = PR[90,2] + 5.794;
   1:  PR[91,3] = PR[90,3] + 4.692;
   1:L PR[91] R[100]mm/sec CNT100;
   1:  PR[91,1] = PR[90,1] + -4.405;
   1:  PR[91,2] = PR[90,2] + 6.677;
   1:  PR[91,3] = PR[90,3] + 4.696;
   1:L PR[91] R[100]mm/sec CNT100;
   1:  PR[91,1] = PR[90,1] + -4.708;
   1:  PR[91,2] = PR[90,2] + 7.390;
   1:  PR[91,3] = PR[90,3] + 4.702;
   1:L PR[91] R[100]mm/sec CNT100;
   1:  PR[91,1] = PR[90,1] + -5.043;
   1:  PR[91,2] = PR[90,2] + 8.088;
   1:  PR[91,3] = PR[90,3] + 4.707;
   1:L PR[91] R[100]mm/sec CNT100;
   1:  PR[91,1] = PR[90,1] + -5.408;
   1:  PR[91,2] = PR[90,2] + 8.766;
   1:  PR[91,3] = PR[90,3] + 4.711;
   1:L PR[91] R[100]mm/sec CNT100;
   1:  PR[91,1] = PR[90,1] + -5.898;
   1:  PR[91,2] = PR[90,2] + 9.578;
   1:  PR[91,3] = PR[90,3] + 4.716;
   1:L PR[91] R[100]mm/sec CNT100;
   1:  PR[91,1] = PR[90,1] + -6.328;
   1:  PR[91,2] = PR[90,2] + 10.213;
   1:  PR[91,3] = PR[90,3] + 4.722;
   1:L PR[91] R[100]mm/sec CNT100;
   1:  PR[91,1] = PR[90,1] + -6.902;
   1:  PR[91,2] = PR[90,2] + 10.974;
   1:  PR[91,3] = PR[90,3] + 4.726;
   1:L PR[91] R[100]mm/sec CNT100;
   1:  PR[91,1] = PR[90,1] + -7.392;
   1:  PR[91,2] = PR[90,2] + 11.561;
   1:  PR[91,3] = PR[90,3] + 4.732;
   1:L PR[91] R[100]mm/sec CNT100;
   1:  PR[91,1] = PR[90,1] + -8.046;
   1:  PR[91,2] = PR[90,2] + 12.264;
   1:  PR[91,3] = PR[90,3] + 4.737;
   1:L PR[91] R[100]mm/sec CNT100;
   1:  PR[91,1] = PR[90,1] + -8.593;
   1:  PR[91,2] = PR[90,2] + 12.798;
   1:  PR[91,3] = PR[90,3] + 4.743;
   1:L PR[91] R[100]mm/sec CNT100;
   1:  PR[91,1] = PR[90,1] + -9.163;
   1:  PR[91,2] = PR[90,2] + 13.305;
   1:  PR[91,3] = PR[90,3] + 4.747;
   1:L PR[91] R[100]mm/sec CNT100;
   1:  PR[91,1] = PR[90,1] + -9.752;
   1:  PR[91,2] = PR[90,2] + 13.783;
   1:  PR[91,3] = PR[90,3] + 4.752;
   1:L PR[91] R[100]mm/sec CNT100;
   1:  PR[91,1] = PR[90,1] + -10.360;
   1:  PR[91,2] = PR[90,2] + 14.231;
   1:  PR[91,3] = PR[90,3] + 4.757;
   1:L PR[91] R[100]mm/sec CNT100;
   1:  PR[91,1] = PR[90,1] + -11.168;
   1:  PR[91,2] = PR[90,2] + 14.770;
   1:  PR[91,3] = PR[90,3] + 4.761;
   1:L PR[91] R[100]mm/sec CNT100;
   1:  PR[91,1] = PR[90,1] + -11.813;
   1:  PR[91,2] = PR[90,2] + 15.151;
   1:  PR[91,3] = PR[90,3] + 4.767;
   1:L PR[91] R[100]mm/sec CNT100;
   1:  PR[91,1] = PR[90,1] + -12.679;
   1:  PR[91,2] = PR[90,2] + 15.608;
   1:  PR[91,3] = PR[90,3] + 4.772;
   1:L PR[91] R[100]mm/sec CNT100;
   1:  PR[91,1] = PR[90,1] + -13.358;
   1:  PR[91,2] = PR[90,2] + 15.921;
   1:  PR[91,3] = PR[90,3] + 4.778;
   1:L PR[91] R[100]mm/sec CNT100;
   1:  PR[91,1] = PR[90,1] + -14.273;
   1:  PR[91,2] = PR[90,2] + 16.289;
   1:  PR[91,3] = PR[90,3] + 4.782;
   1:L PR[91] R[100]mm/sec CNT100;
   1:  PR[91,1] = PR[90,1] + -14.979;
   1:  PR[91,2] = PR[90,2] + 16.531;
   1:  PR[91,3] = PR[90,3] + 4.788;
   1:L PR[91] R[100]mm/sec CNT100;
   1:  PR[91,1] = PR[90,1] + -15.693;
   1:  PR[91,2] = PR[90,2] + 16.741;
   1:  PR[91,3] = PR[90,3] + 4.793;
   1:L PR[91] R[100]mm/sec CNT100;
   1:  PR[91,1] = PR[90,1] + -16.661;
   1:  PR[91,2] = PR[90,2] + 16.973;
   1:  PR[91,3] = PR[90,3] + 4.797;
   1:L PR[91] R[100]mm/sec CNT100;
   1:  PR[91,1] = PR[90,1] + -17.387;
   1:  PR[91,2] = PR[90,2] + 17.108;
   1:  PR[91,3] = PR[90,3] + 4.803;
   1:L PR[91] R[100]mm/sec CNT100;
   1:  PR[91,1] = PR[90,1] + -18.381;
   1:  PR[91,2] = PR[90,2] + 17.239;
   1:  PR[91,3] = PR[90,3] + 4.808;
   1:L PR[91] R[100]mm/sec CNT100;
   1:  PR[91,1] = PR[90,1] + -19.118;
   1:  PR[91,2] = PR[90,2] + 17.300;
   1:  PR[91,3] = PR[90,3] + 4.814;
   1:L PR[91] R[100]mm/sec CNT100;
   1:  PR[91,1] = PR[90,1] + -19.853;
   1:  PR[91,2] = PR[90,2] + 17.327;
   1:  PR[91,3] = PR[90,3] + 4.818;
   1:L PR[91] R[100]mm/sec CNT100;
   1:  PR[91,1] = PR[90,1] + -20.864;
   1:  PR[91,2] = PR[90,2] + 17.312;
   1:  PR[91,3] = PR[90,3] + 4.823;
   1:L PR[91] R[100]mm/sec CNT100;
   1:  PR[91,1] = PR[90,1] + -21.596;
   1:  PR[91,2] = PR[90,2] + 17.263;
   1:  PR[91,3] = PR[90,3] + 4.829;
   1:L PR[91] R[100]mm/sec CNT100;
   1:  PR[91,1] = PR[90,1] + -22.322;
   1:  PR[91,2] = PR[90,2] + 17.183;
   1:  PR[91,3] = PR[90,3] + 4.833;
   1:L PR[91] R[100]mm/sec CNT100;
   1:  PR[91,1] = PR[90,1] + -23.324;
   1:  PR[91,2] = PR[90,2] + 17.020;
   1:  PR[91,3] = PR[90,3] + 4.838;
   1:L PR[91] R[100]mm/sec CNT100;
   1:  PR[91,1] = PR[90,1] + -24.323;
   1:  PR[91,2] = PR[90,2] + 16.793;
   1:  PR[91,3] = PR[90,3] + 4.844;
   1:L PR[91] R[100]mm/sec CNT100;
   1:  PR[91,1] = PR[90,1] + -24.742;
   1:  PR[91,2] = PR[90,2] + 16.681;
   1:  PR[91,3] = PR[90,3] + 4.850;
   1:L PR[91] R[100]mm/sec CNT100;
   1:  PR[91,1] = PR[90,1] + -25.435;
   1:  PR[91,2] = PR[90,2] + 16.466;
   1:  PR[91,3] = PR[90,3] + 4.853;
   1:L PR[91] R[100]mm/sec CNT100;
   1:  PR[91,1] = PR[90,1] + -26.397;
   1:  PR[91,2] = PR[90,2] + 16.116;
   1:  PR[91,3] = PR[90,3] + 4.857;
   1:L PR[91] R[100]mm/sec CNT100;
   1:  PR[91,1] = PR[90,1] + -27.338;
   1:  PR[91,2] = PR[90,2] + 15.705;
   1:  PR[91,3] = PR[90,3] + 4.863;
   1:L PR[91] R[100]mm/sec CNT100;
   1:  PR[91,1] = PR[90,1] + -27.985;
   1:  PR[91,2] = PR[90,2] + 15.383;
   1:  PR[91,3] = PR[90,3] + 4.870;
   1:L PR[91] R[100]mm/sec CNT100;
   1:  PR[91,1] = PR[90,1] + -28.617;
   1:  PR[91,2] = PR[90,2] + 15.032;
   1:  PR[91,3] = PR[90,3] + 4.874;
   1:L PR[91] R[100]mm/sec CNT100;
   1:  PR[91,1] = PR[90,1] + -29.230;
   1:  PR[91,2] = PR[90,2] + 14.657;
   1:  PR[91,3] = PR[90,3] + 4.878;
   1:L PR[91] R[100]mm/sec CNT100;
   1:  PR[91,1] = PR[90,1] + -30.084;
   1:  PR[91,2] = PR[90,2] + 14.073;
   1:  PR[91,3] = PR[90,3] + 4.883;
   1:L PR[91] R[100]mm/sec CNT100;
   1:  PR[91,1] = PR[90,1] + -30.902;
   1:  PR[91,2] = PR[90,2] + 13.435;
   1:  PR[91,3] = PR[90,3] + 4.889;
   1:L PR[91] R[100]mm/sec CNT100;
   1:  PR[91,1] = PR[90,1] + -31.445;
   1:  PR[91,2] = PR[90,2] + 12.966;
   1:  PR[91,3] = PR[90,3] + 4.895;
   1:L PR[91] R[100]mm/sec CNT100;
   1:  PR[91,1] = PR[90,1] + -31.967;
   1:  PR[91,2] = PR[90,2] + 12.473;
   1:  PR[91,3] = PR[90,3] + 4.900;
   1:L PR[91] R[100]mm/sec CNT100;
   1:  PR[91,1] = PR[90,1] + -32.465;
   1:  PR[91,2] = PR[90,2] + 11.961;
   1:  PR[91,3] = PR[90,3] + 4.904;
   1:L PR[91] R[100]mm/sec CNT100;
   1:  PR[91,1] = PR[90,1] + -33.153;
   1:  PR[91,2] = PR[90,2] + 11.178;
   1:  PR[91,3] = PR[90,3] + 4.909;
   1:L PR[91] R[100]mm/sec CNT100;
   1:  PR[91,1] = PR[90,1] + -33.791;
   1:  PR[91,2] = PR[90,2] + 10.351;
   1:  PR[91,3] = PR[90,3] + 4.915;
   1:L PR[91] R[100]mm/sec CNT100;
   1:  PR[91,1] = PR[90,1] + -34.200;
   1:  PR[91,2] = PR[90,2] + 9.764;
   1:  PR[91,3] = PR[90,3] + 4.921;
   1:L PR[91] R[100]mm/sec CNT100;
   1:  PR[91,1] = PR[90,1] + -34.404;
   1:  PR[91,2] = PR[90,2] + 9.445;
   1:  PR[91,3] = PR[90,3] + 4.926;
   1:L PR[91] R[100]mm/sec CNT100;
   1:  PR[91,1] = PR[90,1] + -34.938;
   1:  PR[91,2] = PR[90,2] + 8.541;
   1:  PR[91,3] = PR[90,3] + 4.928;
   1:L PR[91] R[100]mm/sec CNT100;
   1:  PR[91,1] = PR[90,1] + -35.411;
   1:  PR[91,2] = PR[90,2] + 7.611;
   1:  PR[91,3] = PR[90,3] + 4.934;
   1:L PR[91] R[100]mm/sec CNT100;
   1:  PR[91,1] = PR[90,1] + -35.827;
   1:  PR[91,2] = PR[90,2] + 6.643;
   1:  PR[91,3] = PR[90,3] + 4.941;
   1:L PR[91] R[100]mm/sec CNT100;
   1:  PR[91,1] = PR[90,1] + -35.961;
   1:  PR[91,2] = PR[90,2] + 6.297;
   1:  PR[91,3] = PR[90,3] + 4.947;
   1:L PR[91] R[100]mm/sec CNT100;
   1:  PR[91,1] = PR[90,1] + -36.193;
   1:  PR[91,2] = PR[90,2] + 5.624;
   1:  PR[91,3] = PR[90,3] + 4.949;
   1:L PR[91] R[100]mm/sec CNT100;
   1:  PR[91,1] = PR[90,1] + -36.486;
   1:  PR[91,2] = PR[90,2] + 4.616;
   1:  PR[91,3] = PR[90,3] + 4.954;
   1:L PR[91] R[100]mm/sec CNT100;
   1:  PR[91,1] = PR[90,1] + -36.714;
   1:  PR[91,2] = PR[90,2] + 3.591;
   1:  PR[91,3] = PR[90,3] + 4.960;
   1:L PR[91] R[100]mm/sec CNT100;
   1:  PR[91,1] = PR[90,1] + -36.833;
   1:  PR[91,2] = PR[90,2] + 2.892;
   1:  PR[91,3] = PR[90,3] + 4.966;
   1:L PR[91] R[100]mm/sec CNT100;
   1:  PR[91,1] = PR[90,1] + -36.922;
   1:  PR[91,2] = PR[90,2] + 2.188;
   1:  PR[91,3] = PR[90,3] + 4.971;
   1:L PR[91] R[100]mm/sec CNT100;
   1:  PR[91,1] = PR[90,1] + -36.998;
   1:  PR[91,2] = PR[90,2] + 1.140;
   1:  PR[91,3] = PR[90,3] + 4.975;
   1:L PR[91] R[100]mm/sec CNT100;
   1:  PR[91,1] = PR[90,1] + -37.007;
   1:  PR[91,2] = PR[90,2] + 0.083;
   1:  PR[91,3] = PR[90,3] + 4.981;
   1:L PR[91] R[100]mm/sec CNT100;
   1:  PR[91,1] = PR[90,1] + -36.998;
   1:  PR[91,2] = PR[90,2] + -0.283;
   1:  PR[91,3] = PR[90,3] + 4.988;
   1:L PR[91] R[100]mm/sec CNT100;
   1:  PR[91,1] = PR[90,1] + -36.952;
   1:  PR[91,2] = PR[90,2] + -0.992;
   1:  PR[91,3] = PR[90,3] + 4.990;
   1:L PR[91] R[100]mm/sec CNT100;
   1:  PR[91,1] = PR[90,1] + -36.833;
   1:  PR[91,2] = PR[90,2] + -2.040;
   1:  PR[91,3] = PR[90,3] + 4.994;
   1:L PR[91] R[100]mm/sec CNT100;
   1:  PR[91,1] = PR[90,1] + -36.714;
   1:  PR[91,2] = PR[90,2] + -2.736;
   1:  PR[91,3] = PR[90,3] + 5.001;
   1:L PR[91] R[100]mm/sec CNT100;
   1:  PR[91,1] = PR[90,1] + -36.486;
   1:  PR[91,2] = PR[90,2] + -3.764;
   1:  PR[91,3] = PR[90,3] + 5.005;
   1:L PR[91] R[100]mm/sec CNT100;
   1:  PR[91,1] = PR[90,1] + -36.295;
   1:  PR[91,2] = PR[90,2] + -4.447;
   1:  PR[91,3] = PR[90,3] + 5.011;
   1:L PR[91] R[100]mm/sec CNT100;
   1:  PR[91,1] = PR[90,1] + -36.075;
   1:  PR[91,2] = PR[90,2] + -5.123;
   1:  PR[91,3] = PR[90,3] + 5.016;
   1:L PR[91] R[100]mm/sec CNT100;
   1:  PR[91,1] = PR[90,1] + -35.700;
   1:  PR[91,2] = PR[90,2] + -6.106;
   1:  PR[91,3] = PR[90,3] + 5.020;
   1:L PR[91] R[100]mm/sec CNT100;
   1:  PR[91,1] = PR[90,1] + -35.412;
   1:  PR[91,2] = PR[90,2] + -6.752;
   1:  PR[91,3] = PR[90,3] + 5.026;
   1:L PR[91] R[100]mm/sec CNT100;
   1:  PR[91,1] = PR[90,1] + -34.938;
   1:  PR[91,2] = PR[90,2] + -7.686;
   1:  PR[91,3] = PR[90,3] + 5.031;
   1:L PR[91] R[100]mm/sec CNT100;
   1:  PR[91,1] = PR[90,1] + -34.404;
   1:  PR[91,2] = PR[90,2] + -8.590;
   1:  PR[91,3] = PR[90,3] + 5.037;
   1:L PR[91] R[100]mm/sec CNT100;
   1:  PR[91,1] = PR[90,1] + -34.200;
   1:  PR[91,2] = PR[90,2] + -8.909;
   1:  PR[91,3] = PR[90,3] + 5.043;
   1:L PR[91] R[100]mm/sec CNT100;
   1:  PR[91,1] = PR[90,1] + -33.787;
   1:  PR[91,2] = PR[90,2] + -9.502;
   1:  PR[91,3] = PR[90,3] + 5.046;
   1:L PR[91] R[100]mm/sec CNT100;
   1:  PR[91,1] = PR[90,1] + -33.598;
   1:  PR[91,2] = PR[90,2] + -9.759;
   1:  PR[91,3] = PR[90,3] + 5.050;
   1:L PR[91] R[100]mm/sec CNT100;
   1:  PR[91,1] = PR[90,1] + -33.153;
   1:  PR[91,2] = PR[90,2] + -10.323;
   1:  PR[91,3] = PR[90,3] + 5.052;
   1:L PR[91] R[100]mm/sec CNT100;
   1:  PR[91,1] = PR[90,1] + -32.687;
   1:  PR[91,2] = PR[90,2] + -10.864;
   1:  PR[91,3] = PR[90,3] + 5.056;
   1:L PR[91] R[100]mm/sec CNT100;
   1:  PR[91,1] = PR[90,1] + -31.965;
   1:  PR[91,2] = PR[90,2] + -11.620;
   1:  PR[91,3] = PR[90,3] + 5.061;
   1:L PR[91] R[100]mm/sec CNT100;
   1:  PR[91,1] = PR[90,1] + -31.445;
   1:  PR[91,2] = PR[90,2] + -12.111;
   1:  PR[91,3] = PR[90,3] + 5.067;
   1:L PR[91] R[100]mm/sec CNT100;
   1:  PR[91,1] = PR[90,1] + -30.901;
   1:  PR[91,2] = PR[90,2] + -12.580;
   1:  PR[91,3] = PR[90,3] + 5.071;
   1:L PR[91] R[100]mm/sec CNT100;
   1:  PR[91,1] = PR[90,1] + -30.084;
   1:  PR[91,2] = PR[90,2] + -13.218;
   1:  PR[91,3] = PR[90,3] + 5.076;
   1:L PR[91] R[100]mm/sec CNT100;
   1:  PR[91,1] = PR[90,1] + -29.230;
   1:  PR[91,2] = PR[90,2] + -13.801;
   1:  PR[91,3] = PR[90,3] + 5.082;
   1:L PR[91] R[100]mm/sec CNT100;
   1:  PR[91,1] = PR[90,1] + -28.617;
   1:  PR[91,2] = PR[90,2] + -14.177;
   1:  PR[91,3] = PR[90,3] + 5.088;
   1:L PR[91] R[100]mm/sec CNT100;
   1:  PR[91,1] = PR[90,1] + -27.988;
   1:  PR[91,2] = PR[90,2] + -14.526;
   1:  PR[91,3] = PR[90,3] + 5.093;
   1:L PR[91] R[100]mm/sec CNT100;
   1:  PR[91,1] = PR[90,1] + -27.060;
   1:  PR[91,2] = PR[90,2] + -14.978;
   1:  PR[91,3] = PR[90,3] + 5.097;
   1:L PR[91] R[100]mm/sec CNT100;
   1:  PR[91,1] = PR[90,1] + -26.396;
   1:  PR[91,2] = PR[90,2] + -15.262;
   1:  PR[91,3] = PR[90,3] + 5.103;
   1:L PR[91] R[100]mm/sec CNT100;
   1:  PR[91,1] = PR[90,1] + -25.719;
   1:  PR[91,2] = PR[90,2] + -15.516;
   1:  PR[91,3] = PR[90,3] + 5.108;
   1:L PR[91] R[100]mm/sec CNT100;
   1:  PR[91,1] = PR[90,1] + -24.741;
   1:  PR[91,2] = PR[90,2] + -15.826;
   1:  PR[91,3] = PR[90,3] + 5.112;
   1:L PR[91] R[100]mm/sec CNT100;
   1:  PR[91,1] = PR[90,1] + -24.039;
   1:  PR[91,2] = PR[90,2] + -16.011;
   1:  PR[91,3] = PR[90,3] + 5.118;
   1:L PR[91] R[100]mm/sec CNT100;
   1:  PR[91,1] = PR[90,1] + -23.327;
   1:  PR[91,2] = PR[90,2] + -16.165;
   1:  PR[91,3] = PR[90,3] + 5.123;
   1:L PR[91] R[100]mm/sec CNT100;
   1:  PR[91,1] = PR[90,1] + -22.322;
   1:  PR[91,2] = PR[90,2] + -16.328;
   1:  PR[91,3] = PR[90,3] + 5.127;
   1:L PR[91] R[100]mm/sec CNT100;
   1:  PR[91,1] = PR[90,1] + -21.596;
   1:  PR[91,2] = PR[90,2] + -16.408;
   1:  PR[91,3] = PR[90,3] + 5.133;
   1:L PR[91] R[100]mm/sec CNT100;
   1:  PR[91,1] = PR[90,1] + -20.864;
   1:  PR[91,2] = PR[90,2] + -16.456;
   1:  PR[91,3] = PR[90,3] + 5.138;
   1:L PR[91] R[100]mm/sec CNT100;
   1:  PR[91,1] = PR[90,1] + -19.853;
   1:  PR[91,2] = PR[90,2] + -16.471;
   1:  PR[91,3] = PR[90,3] + 5.142;
   1:L PR[91] R[100]mm/sec CNT100;
   1:  PR[91,1] = PR[90,1] + -19.118;
   1:  PR[91,2] = PR[90,2] + -16.444;
   1:  PR[91,3] = PR[90,3] + 5.148;
   1:L PR[91] R[100]mm/sec CNT100;
   1:  PR[91,1] = PR[90,1] + -18.382;
   1:  PR[91,2] = PR[90,2] + -16.384;
   1:  PR[91,3] = PR[90,3] + 5.153;
   1:L PR[91] R[100]mm/sec CNT100;
   1:  PR[91,1] = PR[90,1] + -17.387;
   1:  PR[91,2] = PR[90,2] + -16.253;
   1:  PR[91,3] = PR[90,3] + 5.157;
   1:L PR[91] R[100]mm/sec CNT100;
   1:  PR[91,1] = PR[90,1] + -16.661;
   1:  PR[91,2] = PR[90,2] + -16.118;
   1:  PR[91,3] = PR[90,3] + 5.163;
   1:L PR[91] R[100]mm/sec CNT100;
   1:  PR[91,1] = PR[90,1] + -15.693;
   1:  PR[91,2] = PR[90,2] + -15.886;
   1:  PR[91,3] = PR[90,3] + 5.168;
   1:L PR[91] R[100]mm/sec CNT100;
   1:  PR[91,1] = PR[90,1] + -14.980;
   1:  PR[91,2] = PR[90,2] + -15.676;
   1:  PR[91,3] = PR[90,3] + 5.174;
   1:L PR[91] R[100]mm/sec CNT100;
   1:  PR[91,1] = PR[90,1] + -14.272;
   1:  PR[91,2] = PR[90,2] + -15.433;
   1:  PR[91,3] = PR[90,3] + 5.179;
   1:L PR[91] R[100]mm/sec CNT100;
   1:  PR[91,1] = PR[90,1] + -13.573;
   1:  PR[91,2] = PR[90,2] + -15.157;
   1:  PR[91,3] = PR[90,3] + 5.183;
   1:L PR[91] R[100]mm/sec CNT100;
   1:  PR[91,1] = PR[90,1] + -12.678;
   1:  PR[91,2] = PR[90,2] + -14.752;
   1:  PR[91,3] = PR[90,3] + 5.188;
   1:L PR[91] R[100]mm/sec CNT100;
   1:  PR[91,1] = PR[90,1] + -11.813;
   1:  PR[91,2] = PR[90,2] + -14.296;
   1:  PR[91,3] = PR[90,3] + 5.194;
   1:L PR[91] R[100]mm/sec CNT100;
   1:  PR[91,1] = PR[90,1] + -11.166;
   1:  PR[91,2] = PR[90,2] + -13.913;
   1:  PR[91,3] = PR[90,3] + 5.200;
   1:L PR[91] R[100]mm/sec CNT100;
   1:  PR[91,1] = PR[90,1] + -10.535;
   1:  PR[91,2] = PR[90,2] + -13.500;
   1:  PR[91,3] = PR[90,3] + 5.204;
   1:L PR[91] R[100]mm/sec CNT100;
   1:  PR[91,1] = PR[90,1] + -9.752;
   1:  PR[91,2] = PR[90,2] + -12.927;
   1:  PR[91,3] = PR[90,3] + 5.209;
   1:L PR[91] R[100]mm/sec CNT100;
   1:  PR[91,1] = PR[90,1] + -9.163;
   1:  PR[91,2] = PR[90,2] + -12.450;
   1:  PR[91,3] = PR[90,3] + 5.215;
   1:L PR[91] R[100]mm/sec CNT100;
   1:  PR[91,1] = PR[90,1] + -8.593;
   1:  PR[91,2] = PR[90,2] + -11.943;
   1:  PR[91,3] = PR[90,3] + 5.219;
   1:L PR[91] R[100]mm/sec CNT100;
   1:  PR[91,1] = PR[90,1] + -8.046;
   1:  PR[91,2] = PR[90,2] + -11.409;
   1:  PR[91,3] = PR[90,3] + 5.224;
   1:L PR[91] R[100]mm/sec CNT100;
   1:  PR[91,1] = PR[90,1] + -7.392;
   1:  PR[91,2] = PR[90,2] + -10.706;
   1:  PR[91,3] = PR[90,3] + 5.228;
   1:L PR[91] R[100]mm/sec CNT100;
   1:  PR[91,1] = PR[90,1] + -6.902;
   1:  PR[91,2] = PR[90,2] + -10.119;
   1:  PR[91,3] = PR[90,3] + 5.234;
   1:L PR[91] R[100]mm/sec CNT100;
   1:  PR[91,1] = PR[90,1] + -6.328;
   1:  PR[91,2] = PR[90,2] + -9.357;
   1:  PR[91,3] = PR[90,3] + 5.239;
   1:L PR[91] R[100]mm/sec CNT100;
   1:  PR[91,1] = PR[90,1] + -5.898;
   1:  PR[91,2] = PR[90,2] + -8.721;
   1:  PR[91,3] = PR[90,3] + 5.245;
   1:L PR[91] R[100]mm/sec CNT100;
   1:  PR[91,1] = PR[90,1] + -5.495;
   1:  PR[91,2] = PR[90,2] + -8.063;
   1:  PR[91,3] = PR[90,3] + 5.249;
   1:L PR[91] R[100]mm/sec CNT100;
   1:  PR[91,1] = PR[90,1] + -5.043;
   1:  PR[91,2] = PR[90,2] + -7.234;
   1:  PR[91,3] = PR[90,3] + 5.254;
   1:L PR[91] R[100]mm/sec CNT100;
   1:  PR[91,1] = PR[90,1] + -4.642;
   1:  PR[91,2] = PR[90,2] + -6.383;
   1:  PR[91,3] = PR[90,3] + 5.260;
   1:L PR[91] R[100]mm/sec CNT100;
   1:  PR[91,1] = PR[90,1] + -4.345;
   1:  PR[91,2] = PR[90,2] + -5.669;
   1:  PR[91,3] = PR[90,3] + 5.266;
   1:L PR[91] R[100]mm/sec CNT100;
   1:  PR[91,1] = PR[90,1] + -4.136;
   1:  PR[91,2] = PR[90,2] + -5.095;
   1:  PR[91,3] = PR[90,3] + 5.270;
   1:L PR[91] R[100]mm/sec CNT100;
   1:  PR[91,1] = PR[90,1] + -3.810;
   1:  PR[91,2] = PR[90,2] + -4.043;
   1:  PR[91,3] = PR[90,3] + 5.274;
   1:L PR[91] R[100]mm/sec CNT100;
   1:  PR[91,1] = PR[90,1] + -3.621;
   1:  PR[91,2] = PR[90,2] + -3.289;
   1:  PR[91,3] = PR[90,3] + 5.281;
   1:L PR[91] R[100]mm/sec CNT100;
   1:  PR[91,1] = PR[90,1] + -3.387;
   1:  PR[91,2] = PR[90,2] + -2.191;
   1:  PR[91,3] = PR[90,3] + 5.285;
   1:L PR[91] R[100]mm/sec CNT100;
   1:  PR[91,1] = PR[90,1] + -3.231;
   1:  PR[91,2] = PR[90,2] + -1.778;
   1:  PR[91,3] = PR[90,3] + 5.292;
   1:L PR[91] R[100]mm/sec CNT100;
   1:  PR[91,1] = PR[90,1] + -3.063;
   1:  PR[91,2] = PR[90,2] + -1.462;
   1:  PR[91,3] = PR[90,3] + 5.295;
   1:L PR[91] R[100]mm/sec CNT100;
   1:  PR[91,1] = PR[90,1] + -2.860;
   1:  PR[91,2] = PR[90,2] + -1.170;
   1:  PR[91,3] = PR[90,3] + 5.297;
   1:L PR[91] R[100]mm/sec CNT100;
   1:  PR[91,1] = PR[90,1] + -2.570;
   1:  PR[91,2] = PR[90,2] + -0.844;
   1:  PR[91,3] = PR[90,3] + 5.299;
   1:L PR[91] R[100]mm/sec CNT100;
   1:  PR[91,1] = PR[90,1] + -2.235;
   1:  PR[91,2] = PR[90,2] + -0.563;
   1:  PR[91,3] = PR[90,3] + 5.302;
   1:L PR[91] R[100]mm/sec CNT100;
   1:  PR[91,1] = PR[90,1] + -1.929;
   1:  PR[91,2] = PR[90,2] + -0.367;
   1:  PR[91,3] = PR[90,3] + 5.305;
   1:L PR[91] R[100]mm/sec CNT100;
   1:  PR[91,1] = PR[90,1] + -1.541;
   1:  PR[91,2] = PR[90,2] + -0.184;
   1:  PR[91,3] = PR[90,3] + 5.307;
   1:L PR[91] R[100]mm/sec CNT100;
   1:  PR[91,1] = PR[90,1] + -1.194;
   1:  PR[91,2] = PR[90,2] + -0.071;
   1:  PR[91,3] = PR[90,3] + 5.309;
   1:L PR[91] R[100]mm/sec CNT100;
   1:  PR[91,1] = PR[90,1] + -0.775;
   1:  PR[91,2] = PR[90,2] + 0.007;
   1:  PR[91,3] = PR[90,3] + 5.312;
   1:L PR[91] R[100]mm/sec CNT100;
   1:  PR[91,1] = PR[90,1] + -0.430;
   1:  PR[91,2] = PR[90,2] + 0.028;
   1:  PR[91,3] = PR[90,3] + 5.314;
   1:L PR[91] R[100]mm/sec CNT100;
   1:  PR[91,1] = PR[90,1] + 0.192;
   1:  PR[91,3] = PR[90,3] + 5.316;
   1:L PR[91] R[100]mm/sec CNT100;
   1:  PR[91] = PR[90];
   1:  PR[91,1] = PR[90,1] + 0.483;
   1:  PR[91,2] = PR[90,2] + 0.004;
   1:  PR[91,3] = PR[90,3] + 6.650;
   1:L PR[91] R[100]mm/sec CNT100;
   1:  PR[91,1] = PR[90,1] + 0.870;
   1:  PR[91,2] = PR[90,2] + -0.070;
   1:  PR[91,3] = PR[90,3] + 5.322;
   1:L PR[91] R[100]mm/sec CNT100;
   1:  PR[91,1] = PR[90,1] + 1.245;
   1:  PR[91,2] = PR[90,2] + -0.193;
   1:  PR[91,3] = PR[90,3] + 5.325;
   1:L PR[91] R[100]mm/sec CNT100;
   1:  PR[91,1] = PR[90,1] + 1.602;
   1:  PR[91,2] = PR[90,2] + -0.361;
   1:  PR[91,3] = PR[90,3] + 5.327;
   1:L PR[91] R[100]mm/sec CNT100;
   1:  PR[91,1] = PR[90,1] + 1.934;
   1:  PR[91,2] = PR[90,2] + -0.573;
   1:  PR[91,3] = PR[90,3] + 5.329;
   1:L PR[91] R[100]mm/sec CNT100;
   1:  PR[91,1] = PR[90,1] + 2.236;
   1:  PR[91,2] = PR[90,2] + -0.826;
   1:  PR[91,3] = PR[90,3] + 5.332;
   1:L PR[91] R[100]mm/sec CNT100;
   1:  PR[91,1] = PR[90,1] + 2.505;
   1:  PR[91,2] = PR[90,2] + -1.114;
   1:  PR[91,3] = PR[90,3] + 5.334;
   1:L PR[91] R[100]mm/sec CNT100;
   1:  PR[91,1] = PR[90,1] + 2.735;
   1:  PR[91,2] = PR[90,2] + -1.435;
   1:  PR[91,3] = PR[90,3] + 5.337;
   1:L PR[91] R[100]mm/sec CNT100;
   1:  PR[91,1] = PR[90,1] + 2.923;
   1:  PR[91,2] = PR[90,2] + -1.786;
   1:  PR[91,3] = PR[90,3] + 5.339;
   1:L PR[91] R[100]mm/sec CNT100;
   1:  PR[91,1] = PR[90,1] + 3.068;
   1:  PR[91,2] = PR[90,2] + -2.169;
   1:  PR[91,3] = PR[90,3] + 5.341;
   1:L PR[91] R[100]mm/sec CNT100;
   1:  PR[91,1] = PR[90,1] + 3.318;
   1:  PR[91,2] = PR[90,2] + -3.346;
   1:  PR[91,3] = PR[90,3] + 5.344;
   1:L PR[91] R[100]mm/sec CNT100;
   1:  PR[91,1] = PR[90,1] + 3.526;
   1:  PR[91,2] = PR[90,2] + -4.157;
   1:  PR[91,3] = PR[90,3] + 5.351;
   1:L PR[91] R[100]mm/sec CNT100;
   1:  PR[91,1] = PR[90,1] + 3.773;
   1:  PR[91,2] = PR[90,2] + -4.955;
   1:  PR[91,3] = PR[90,3] + 5.356;
   1:L PR[91] R[100]mm/sec CNT100;
   1:  PR[91,1] = PR[90,1] + 4.060;
   1:  PR[91,2] = PR[90,2] + -5.739;
   1:  PR[91,3] = PR[90,3] + 5.361;
   1:L PR[91] R[100]mm/sec CNT100;
   1:  PR[91,1] = PR[90,1] + 4.385;
   1:  PR[91,2] = PR[90,2] + -6.510;
   1:  PR[91,3] = PR[90,3] + 5.367;
   1:L PR[91] R[100]mm/sec CNT100;
   1:  PR[91,1] = PR[90,1] + 4.748;
   1:  PR[91,2] = PR[90,2] + -7.263;
   1:  PR[91,3] = PR[90,3] + 5.372;
   1:L PR[91] R[100]mm/sec CNT100;
   1:  PR[91,1] = PR[90,1] + 5.148;
   1:  PR[91,2] = PR[90,2] + -7.999;
   1:  PR[91,3] = PR[90,3] + 5.377;
   1:L PR[91] R[100]mm/sec CNT100;
   1:  PR[91,1] = PR[90,1] + 5.584;
   1:  PR[91,2] = PR[90,2] + -8.713;
   1:  PR[91,3] = PR[90,3] + 5.382;
   1:L PR[91] R[100]mm/sec CNT100;
   1:  PR[91,1] = PR[90,1] + 6.055;
   1:  PR[91,2] = PR[90,2] + -9.406;
   1:  PR[91,3] = PR[90,3] + 5.387;
   1:L PR[91] R[100]mm/sec CNT100;
   1:  PR[91,1] = PR[90,1] + 6.559;
   1:  PR[91,2] = PR[90,2] + -10.074;
   1:  PR[91,3] = PR[90,3] + 5.392;
   1:L PR[91] R[100]mm/sec CNT100;
   1:  PR[91,1] = PR[90,1] + 7.096;
   1:  PR[91,2] = PR[90,2] + -10.716;
   1:  PR[91,3] = PR[90,3] + 5.397;
   1:L PR[91] R[100]mm/sec CNT100;
   1:  PR[91,1] = PR[90,1] + 7.664;
   1:  PR[91,2] = PR[90,2] + -11.331;
   1:  PR[91,3] = PR[90,3] + 5.402;
   1:L PR[91] R[100]mm/sec CNT100;
   1:  PR[91,1] = PR[90,1] + 8.261;
   1:  PR[91,2] = PR[90,2] + -11.917;
   1:  PR[91,3] = PR[90,3] + 5.407;
   1:L PR[91] R[100]mm/sec CNT100;
   1:  PR[91,1] = PR[90,1] + 8.901;
   1:  PR[91,2] = PR[90,2] + -12.484;
   1:  PR[91,3] = PR[90,3] + 5.412;
   1:L PR[91] R[100]mm/sec CNT100;
   1:  PR[91,1] = PR[90,1] + 9.540;
   1:  PR[91,2] = PR[90,2] + -12.998;
   1:  PR[91,3] = PR[90,3] + 5.417;
   1:L PR[91] R[100]mm/sec CNT100;
   1:  PR[91,1] = PR[90,1] + 10.218;
   1:  PR[91,2] = PR[90,2] + -13.489;
   1:  PR[91,3] = PR[90,3] + 5.422;
   1:L PR[91] R[100]mm/sec CNT100;
   1:  PR[91,1] = PR[90,1] + 10.918;
   1:  PR[91,2] = PR[90,2] + -13.947;
   1:  PR[91,3] = PR[90,3] + 5.428;
   1:L PR[91] R[100]mm/sec CNT100;
   1:  PR[91,1] = PR[90,1] + 11.640;
   1:  PR[91,2] = PR[90,2] + -14.369;
   1:  PR[91,3] = PR[90,3] + 5.433;
   1:L PR[91] R[100]mm/sec CNT100;
   1:  PR[91,1] = PR[90,1] + 12.383;
   1:  PR[91,2] = PR[90,2] + -14.755;
   1:  PR[91,3] = PR[90,3] + 5.438;
   1:L PR[91] R[100]mm/sec CNT100;
   1:  PR[91,1] = PR[90,1] + 13.143;
   1:  PR[91,2] = PR[90,2] + -15.104;
   1:  PR[91,3] = PR[90,3] + 5.443;
   1:L PR[91] R[100]mm/sec CNT100;
   1:  PR[91,1] = PR[90,1] + 13.920;
   1:  PR[91,2] = PR[90,2] + -15.415;
   1:  PR[91,3] = PR[90,3] + 5.448;
   1:L PR[91] R[100]mm/sec CNT100;
   1:  PR[91,1] = PR[90,1] + 14.711;
   1:  PR[91,2] = PR[90,2] + -15.688;
   1:  PR[91,3] = PR[90,3] + 5.453;
   1:L PR[91] R[100]mm/sec CNT100;
   1:  PR[91,1] = PR[90,1] + 15.515;
   1:  PR[91,2] = PR[90,2] + -15.921;
   1:  PR[91,3] = PR[90,3] + 5.458;
   1:L PR[91] R[100]mm/sec CNT100;
   1:  PR[91,1] = PR[90,1] + 16.329;
   1:  PR[91,2] = PR[90,2] + -16.114;
   1:  PR[91,3] = PR[90,3] + 5.463;
   1:L PR[91] R[100]mm/sec CNT100;
   1:  PR[91,1] = PR[90,1] + 17.152;
   1:  PR[91,2] = PR[90,2] + -16.267;
   1:  PR[91,3] = PR[90,3] + 5.468;
   1:L PR[91] R[100]mm/sec CNT100;
   1:  PR[91,1] = PR[90,1] + 17.981;
   1:  PR[91,2] = PR[90,2] + -16.379;
   1:  PR[91,3] = PR[90,3] + 5.473;
   1:L PR[91] R[100]mm/sec CNT100;
   1:  PR[91,1] = PR[90,1] + 18.815;
   1:  PR[91,2] = PR[90,2] + -16.449;
   1:  PR[91,3] = PR[90,3] + 5.478;
   1:L PR[91] R[100]mm/sec CNT100;
   1:  PR[91,1] = PR[90,1] + 19.651;
   1:  PR[91,2] = PR[90,2] + -16.479;
   1:  PR[91,3] = PR[90,3] + 5.483;
   1:L PR[91] R[100]mm/sec CNT100;
   1:  PR[91,1] = PR[90,1] + 20.488;
   1:  PR[91,2] = PR[90,2] + -16.467;
   1:  PR[91,3] = PR[90,3] + 5.489;
   1:L PR[91] R[100]mm/sec CNT100;
   1:  PR[91,1] = PR[90,1] + 21.322;
   1:  PR[91,2] = PR[90,2] + -16.414;
   1:  PR[91,3] = PR[90,3] + 5.494;
   1:L PR[91] R[100]mm/sec CNT100;
   1:  PR[91,1] = PR[90,1] + 22.154;
   1:  PR[91,2] = PR[90,2] + -16.320;
   1:  PR[91,3] = PR[90,3] + 5.499;
   1:L PR[91] R[100]mm/sec CNT100;
   1:  PR[91,1] = PR[90,1] + 22.979;
   1:  PR[91,2] = PR[90,2] + -16.185;
   1:  PR[91,3] = PR[90,3] + 5.504;
   1:L PR[91] R[100]mm/sec CNT100;
   1:  PR[91,1] = PR[90,1] + 23.797;
   1:  PR[91,2] = PR[90,2] + -16.009;
   1:  PR[91,3] = PR[90,3] + 5.509;
   1:L PR[91] R[100]mm/sec CNT100;
   1:  PR[91,1] = PR[90,1] + 24.605;
   1:  PR[91,2] = PR[90,2] + -15.794;
   1:  PR[91,3] = PR[90,3] + 5.514;
   1:L PR[91] R[100]mm/sec CNT100;
   1:  PR[91,1] = PR[90,1] + 25.401;
   1:  PR[91,2] = PR[90,2] + -15.538;
   1:  PR[91,3] = PR[90,3] + 5.519;
   1:L PR[91] R[100]mm/sec CNT100;
   1:  PR[91,1] = PR[90,1] + 26.184;
   1:  PR[91,2] = PR[90,2] + -15.244;
   1:  PR[91,3] = PR[90,3] + 5.524;
   1:L PR[91] R[100]mm/sec CNT100;
   1:  PR[91,1] = PR[90,1] + 26.952;
   1:  PR[91,2] = PR[90,2] + -14.911;
   1:  PR[91,3] = PR[90,3] + 5.529;
   1:L PR[91] R[100]mm/sec CNT100;
   1:  PR[91,1] = PR[90,1] + 27.701;
   1:  PR[91,2] = PR[90,2] + -14.541;
   1:  PR[91,3] = PR[90,3] + 5.534;
   1:L PR[91] R[100]mm/sec CNT100;
   1:  PR[91,1] = PR[90,1] + 28.432;
   1:  PR[91,2] = PR[90,2] + -14.134;
   1:  PR[91,3] = PR[90,3] + 5.539;
   1:L PR[91] R[100]mm/sec CNT100;
   1:  PR[91,1] = PR[90,1] + 29.141;
   1:  PR[91,2] = PR[90,2] + -13.692;
   1:  PR[91,3] = PR[90,3] + 5.544;
   1:L PR[91] R[100]mm/sec CNT100;
   1:  PR[91,1] = PR[90,1] + 29.828;
   1:  PR[91,2] = PR[90,2] + -13.216;
   1:  PR[91,3] = PR[90,3] + 5.550;
   1:L PR[91] R[100]mm/sec CNT100;
   1:  PR[91,1] = PR[90,1] + 30.491;
   1:  PR[91,2] = PR[90,2] + -12.706;
   1:  PR[91,3] = PR[90,3] + 5.555;
   1:L PR[91] R[100]mm/sec CNT100;
   1:  PR[91,1] = PR[90,1] + 31.127;
   1:  PR[91,2] = PR[90,2] + -12.164;
   1:  PR[91,3] = PR[90,3] + 5.560;
   1:L PR[91] R[100]mm/sec CNT100;
   1:  PR[91,1] = PR[90,1] + 31.736;
   1:  PR[91,2] = PR[90,2] + -11.591;
   1:  PR[91,3] = PR[90,3] + 5.565;
   1:L PR[91] R[100]mm/sec CNT100;
   1:  PR[91,1] = PR[90,1] + 32.316;
   1:  PR[91,2] = PR[90,2] + -10.989;
   1:  PR[91,3] = PR[90,3] + 5.570;
   1:L PR[91] R[100]mm/sec CNT100;
   1:  PR[91,1] = PR[90,1] + 32.865;
   1:  PR[91,2] = PR[90,2] + -10.359;
   1:  PR[91,3] = PR[90,3] + 5.575;
   1:L PR[91] R[100]mm/sec CNT100;
   1:  PR[91,1] = PR[90,1] + 33.382;
   1:  PR[91,2] = PR[90,2] + -9.702;
   1:  PR[91,3] = PR[90,3] + 5.580;
   1:L PR[91] R[100]mm/sec CNT100;
   1:  PR[91,1] = PR[90,1] + 33.866;
   1:  PR[91,2] = PR[90,2] + -9.021;
   1:  PR[91,3] = PR[90,3] + 5.585;
   1:L PR[91] R[100]mm/sec CNT100;
   1:  PR[91,1] = PR[90,1] + 34.316;
   1:  PR[91,2] = PR[90,2] + -8.317;
   1:  PR[91,3] = PR[90,3] + 5.590;
   1:L PR[91] R[100]mm/sec CNT100;
   1:  PR[91,1] = PR[90,1] + 34.731;
   1:  PR[91,2] = PR[90,2] + -7.591;
   1:  PR[91,3] = PR[90,3] + 5.595;
   1:L PR[91] R[100]mm/sec CNT100;
   1:  PR[91,1] = PR[90,1] + 35.109;
   1:  PR[91,2] = PR[90,2] + -6.846;
   1:  PR[91,3] = PR[90,3] + 5.600;
   1:L PR[91] R[100]mm/sec CNT100;
   1:  PR[91,1] = PR[90,1] + 35.450;
   1:  PR[91,2] = PR[90,2] + -6.083;
   1:  PR[91,3] = PR[90,3] + 5.605;
   1:L PR[91] R[100]mm/sec CNT100;
   1:  PR[91,1] = PR[90,1] + 35.753;
   1:  PR[91,2] = PR[90,2] + -5.305;
   1:  PR[91,3] = PR[90,3] + 5.610;
   1:L PR[91] R[100]mm/sec CNT100;
   1:  PR[91,1] = PR[90,1] + 36.017;
   1:  PR[91,2] = PR[90,2] + -4.513;
   1:  PR[91,3] = PR[90,3] + 5.616;
   1:L PR[91] R[100]mm/sec CNT100;
   1:  PR[91,1] = PR[90,1] + 36.242;
   1:  PR[91,2] = PR[90,2] + -3.709;
   1:  PR[91,3] = PR[90,3] + 5.621;
   1:L PR[91] R[100]mm/sec CNT100;
   1:  PR[91,1] = PR[90,1] + 36.426;
   1:  PR[91,2] = PR[90,2] + -2.895;
   1:  PR[91,3] = PR[90,3] + 5.626;
   1:L PR[91] R[100]mm/sec CNT100;
   1:  PR[91,1] = PR[90,1] + 36.570;
   1:  PR[91,2] = PR[90,2] + -2.072;
   1:  PR[91,3] = PR[90,3] + 5.631;
   1:L PR[91] R[100]mm/sec CNT100;
   1:  PR[91,1] = PR[90,1] + 36.673;
   1:  PR[91,2] = PR[90,2] + -1.243;
   1:  PR[91,3] = PR[90,3] + 5.636;
   1:L PR[91] R[100]mm/sec CNT100;
   1:  PR[91,1] = PR[90,1] + 36.735;
   1:  PR[91,2] = PR[90,2] + -0.409;
   1:  PR[91,3] = PR[90,3] + 5.641;
   1:L PR[91] R[100]mm/sec CNT100;
   1:  PR[91,1] = PR[90,1] + 36.757;
   1:  PR[91,2] = PR[90,2] + 0.428;
   1:  PR[91,3] = PR[90,3] + 5.646;
   1:L PR[91] R[100]mm/sec CNT100;
   1:  PR[91,1] = PR[90,1] + 36.735;
   1:  PR[91,2] = PR[90,2] + 1.264;
   1:  PR[91,3] = PR[90,3] + 5.651;
   1:L PR[91] R[100]mm/sec CNT100;
   1:  PR[91,1] = PR[90,1] + 36.673;
   1:  PR[91,2] = PR[90,2] + 2.098;
   1:  PR[91,3] = PR[90,3] + 5.656;
   1:L PR[91] R[100]mm/sec CNT100;
   1:  PR[91,1] = PR[90,1] + 36.570;
   1:  PR[91,2] = PR[90,2] + 2.927;
   1:  PR[91,3] = PR[90,3] + 5.661;
   1:L PR[91] R[100]mm/sec CNT100;
   1:  PR[91,1] = PR[90,1] + 36.426;
   1:  PR[91,2] = PR[90,2] + 3.750;
   1:  PR[91,3] = PR[90,3] + 5.666;
   1:L PR[91] R[100]mm/sec CNT100;
   1:  PR[91,1] = PR[90,1] + 36.242;
   1:  PR[91,2] = PR[90,2] + 4.564;
   1:  PR[91,3] = PR[90,3] + 5.671;
   1:L PR[91] R[100]mm/sec CNT100;
   1:  PR[91,1] = PR[90,1] + 36.017;
   1:  PR[91,2] = PR[90,2] + 5.368;
   1:  PR[91,3] = PR[90,3] + 5.677;
   1:L PR[91] R[100]mm/sec CNT100;
   1:  PR[91,1] = PR[90,1] + 35.753;
   1:  PR[91,2] = PR[90,2] + 6.160;
   1:  PR[91,3] = PR[90,3] + 5.682;
   1:L PR[91] R[100]mm/sec CNT100;
   1:  PR[91,1] = PR[90,1] + 35.450;
   1:  PR[91,2] = PR[90,2] + 6.939;
   1:  PR[91,3] = PR[90,3] + 5.687;
   1:L PR[91] R[100]mm/sec CNT100;
   1:  PR[91,1] = PR[90,1] + 35.109;
   1:  PR[91,2] = PR[90,2] + 7.701;
   1:  PR[91,3] = PR[90,3] + 5.692;
   1:L PR[91] R[100]mm/sec CNT100;
   1:  PR[91,1] = PR[90,1] + 34.731;
   1:  PR[91,2] = PR[90,2] + 8.446;
   1:  PR[91,3] = PR[90,3] + 5.697;
   1:L PR[91] R[100]mm/sec CNT100;
   1:  PR[91,1] = PR[90,1] + 34.316;
   1:  PR[91,2] = PR[90,2] + 9.172;
   1:  PR[91,3] = PR[90,3] + 5.702;
   1:L PR[91] R[100]mm/sec CNT100;
   1:  PR[91,1] = PR[90,1] + 33.866;
   1:  PR[91,2] = PR[90,2] + 9.876;
   1:  PR[91,3] = PR[90,3] + 5.707;
   1:L PR[91] R[100]mm/sec CNT100;
   1:  PR[91,1] = PR[90,1] + 33.382;
   1:  PR[91,2] = PR[90,2] + 10.557;
   1:  PR[91,3] = PR[90,3] + 5.712;
   1:L PR[91] R[100]mm/sec CNT100;
   1:  PR[91,1] = PR[90,1] + 32.865;
   1:  PR[91,2] = PR[90,2] + 11.214;
   1:  PR[91,3] = PR[90,3] + 5.717;
   1:L PR[91] R[100]mm/sec CNT100;
   1:  PR[91,1] = PR[90,1] + 32.316;
   1:  PR[91,2] = PR[90,2] + 11.844;
   1:  PR[91,3] = PR[90,3] + 5.722;
   1:L PR[91] R[100]mm/sec CNT100;
   1:  PR[91,1] = PR[90,1] + 31.736;
   1:  PR[91,2] = PR[90,2] + 12.446;
   1:  PR[91,3] = PR[90,3] + 5.727;
   1:L PR[91] R[100]mm/sec CNT100;
   1:  PR[91,1] = PR[90,1] + 31.127;
   1:  PR[91,2] = PR[90,2] + 13.019;
   1:  PR[91,3] = PR[90,3] + 5.732;
   1:L PR[91] R[100]mm/sec CNT100;
   1:  PR[91,1] = PR[90,1] + 30.491;
   1:  PR[91,2] = PR[90,2] + 13.561;
   1:  PR[91,3] = PR[90,3] + 5.737;
   1:L PR[91] R[100]mm/sec CNT100;
   1:  PR[91,1] = PR[90,1] + 29.828;
   1:  PR[91,2] = PR[90,2] + 14.071;
   1:  PR[91,3] = PR[90,3] + 5.743;
   1:L PR[91] R[100]mm/sec CNT100;
   1:  PR[91,1] = PR[90,1] + 29.141;
   1:  PR[91,2] = PR[90,2] + 14.548;
   1:  PR[91,3] = PR[90,3] + 5.748;
   1:L PR[91] R[100]mm/sec CNT100;
   1:  PR[91,1] = PR[90,1] + 28.432;
   1:  PR[91,2] = PR[90,2] + 14.990;
   1:  PR[91,3] = PR[90,3] + 5.753;
   1:L PR[91] R[100]mm/sec CNT100;
   1:  PR[91,1] = PR[90,1] + 27.701;
   1:  PR[91,2] = PR[90,2] + 15.396;
   1:  PR[91,3] = PR[90,3] + 5.758;
   1:L PR[91] R[100]mm/sec CNT100;
   1:  PR[91,1] = PR[90,1] + 26.952;
   1:  PR[91,2] = PR[90,2] + 15.766;
   1:  PR[91,3] = PR[90,3] + 5.763;
   1:L PR[91] R[100]mm/sec CNT100;
   1:  PR[91,1] = PR[90,1] + 26.184;
   1:  PR[91,2] = PR[90,2] + 16.099;
   1:  PR[91,3] = PR[90,3] + 5.768;
   1:L PR[91] R[100]mm/sec CNT100;
   1:  PR[91,1] = PR[90,1] + 25.402;
   1:  PR[91,2] = PR[90,2] + 16.393;
   1:  PR[91,3] = PR[90,3] + 5.773;
   1:L PR[91] R[100]mm/sec CNT100;
   1:  PR[91,1] = PR[90,1] + 24.605;
   1:  PR[91,2] = PR[90,2] + 16.649;
   1:  PR[91,3] = PR[90,3] + 5.778;
   1:L PR[91] R[100]mm/sec CNT100;
   1:  PR[91,1] = PR[90,1] + 23.797;
   1:  PR[91,2] = PR[90,2] + 16.865;
   1:  PR[91,3] = PR[90,3] + 5.783;
   1:L PR[91] R[100]mm/sec CNT100;
   1:  PR[91,1] = PR[90,1] + 22.979;
   1:  PR[91,2] = PR[90,2] + 17.040;
   1:  PR[91,3] = PR[90,3] + 5.788;
   1:L PR[91] R[100]mm/sec CNT100;
   1:  PR[91,1] = PR[90,1] + 22.154;
   1:  PR[91,2] = PR[90,2] + 17.175;
   1:  PR[91,3] = PR[90,3] + 5.793;
   1:L PR[91] R[100]mm/sec CNT100;
   1:  PR[91,1] = PR[90,1] + 21.322;
   1:  PR[91,2] = PR[90,2] + 17.269;
   1:  PR[91,3] = PR[90,3] + 5.798;
   1:L PR[91] R[100]mm/sec CNT100;
   1:  PR[91,1] = PR[90,1] + 20.488;
   1:  PR[91,2] = PR[90,2] + 17.322;
   1:  PR[91,3] = PR[90,3] + 5.803;
   1:L PR[91] R[100]mm/sec CNT100;
   1:  PR[91,1] = PR[90,1] + 19.651;
   1:  PR[91,2] = PR[90,2] + 17.334;
   1:  PR[91,3] = PR[90,3] + 5.809;
   1:L PR[91] R[100]mm/sec CNT100;
   1:  PR[91,1] = PR[90,1] + 18.815;
   1:  PR[91,2] = PR[90,2] + 17.305;
   1:  PR[91,3] = PR[90,3] + 5.814;
   1:L PR[91] R[100]mm/sec CNT100;
   1:  PR[91,1] = PR[90,1] + 17.981;
   1:  PR[91,2] = PR[90,2] + 17.234;
   1:  PR[91,3] = PR[90,3] + 5.819;
   1:L PR[91] R[100]mm/sec CNT100;
   1:  PR[91,1] = PR[90,1] + 17.152;
   1:  PR[91,2] = PR[90,2] + 17.122;
   1:  PR[91,3] = PR[90,3] + 5.824;
   1:L PR[91] R[100]mm/sec CNT100;
   1:  PR[91,1] = PR[90,1] + 16.329;
   1:  PR[91,2] = PR[90,2] + 16.969;
   1:  PR[91,3] = PR[90,3] + 5.829;
   1:L PR[91] R[100]mm/sec CNT100;
   1:  PR[91,1] = PR[90,1] + 15.515;
   1:  PR[91,2] = PR[90,2] + 16.776;
   1:  PR[91,3] = PR[90,3] + 5.834;
   1:L PR[91] R[100]mm/sec CNT100;
   1:  PR[91,1] = PR[90,1] + 14.711;
   1:  PR[91,2] = PR[90,2] + 16.543;
   1:  PR[91,3] = PR[90,3] + 5.839;
   1:L PR[91] R[100]mm/sec CNT100;
   1:  PR[91,1] = PR[90,1] + 13.920;
   1:  PR[91,2] = PR[90,2] + 16.271;
   1:  PR[91,3] = PR[90,3] + 5.844;
   1:L PR[91] R[100]mm/sec CNT100;
   1:  PR[91,1] = PR[90,1] + 13.143;
   1:  PR[91,2] = PR[90,2] + 15.959;
   1:  PR[91,3] = PR[90,3] + 5.849;
   1:L PR[91] R[100]mm/sec CNT100;
   1:  PR[91,1] = PR[90,1] + 12.383;
   1:  PR[91,2] = PR[90,2] + 15.610;
   1:  PR[91,3] = PR[90,3] + 5.854;
   1:L PR[91] R[100]mm/sec CNT100;
   1:  PR[91,1] = PR[90,1] + 11.641;
   1:  PR[91,2] = PR[90,2] + 15.224;
   1:  PR[91,3] = PR[90,3] + 5.859;
   1:L PR[91] R[100]mm/sec CNT100;
   1:  PR[91,1] = PR[90,1] + 10.918;
   1:  PR[91,2] = PR[90,2] + 14.802;
   1:  PR[91,3] = PR[90,3] + 5.865;
   1:L PR[91] R[100]mm/sec CNT100;
   1:  PR[91,1] = PR[90,1] + 10.218;
   1:  PR[91,2] = PR[90,2] + 14.344;
   1:  PR[91,3] = PR[90,3] + 5.870;
   1:L PR[91] R[100]mm/sec CNT100;
   1:  PR[91,1] = PR[90,1] + 9.539;
   1:  PR[91,2] = PR[90,2] + 13.852;
   1:  PR[91,3] = PR[90,3] + 5.875;
   1:L PR[91] R[100]mm/sec CNT100;
   1:  PR[91,1] = PR[90,1] + 8.887;
   1:  PR[91,2] = PR[90,2] + 13.328;
   1:  PR[91,3] = PR[90,3] + 5.880;
   1:L PR[91] R[100]mm/sec CNT100;
   1:  PR[91,1] = PR[90,1] + 8.261;
   1:  PR[91,2] = PR[90,2] + 12.772;
   1:  PR[91,3] = PR[90,3] + 5.885;
   1:L PR[91] R[100]mm/sec CNT100;
   1:  PR[91,1] = PR[90,1] + 7.664;
   1:  PR[91,2] = PR[90,2] + 12.186;
   1:  PR[91,3] = PR[90,3] + 5.890;
   1:L PR[91] R[100]mm/sec CNT100;
   1:  PR[91,1] = PR[90,1] + 7.096;
   1:  PR[91,2] = PR[90,2] + 11.571;
   1:  PR[91,3] = PR[90,3] + 5.895;
   1:L PR[91] R[100]mm/sec CNT100;
   1:  PR[91,1] = PR[90,1] + 6.559;
   1:  PR[91,2] = PR[90,2] + 10.929;
   1:  PR[91,3] = PR[90,3] + 5.900;
   1:L PR[91] R[100]mm/sec CNT100;
   1:  PR[91,1] = PR[90,1] + 6.055;
   1:  PR[91,2] = PR[90,2] + 10.261;
   1:  PR[91,3] = PR[90,3] + 5.905;
   1:L PR[91] R[100]mm/sec CNT100;
   1:  PR[91,1] = PR[90,1] + 5.584;
   1:  PR[91,2] = PR[90,2] + 9.568;
   1:  PR[91,3] = PR[90,3] + 5.910;
   1:L PR[91] R[100]mm/sec CNT100;
   1:  PR[91,1] = PR[90,1] + 5.148;
   1:  PR[91,2] = PR[90,2] + 8.854;
   1:  PR[91,3] = PR[90,3] + 5.915;
   1:L PR[91] R[100]mm/sec CNT100;
   1:  PR[91,1] = PR[90,1] + 4.748;
   1:  PR[91,2] = PR[90,2] + 8.119;
   1:  PR[91,3] = PR[90,3] + 5.920;
   1:L PR[91] R[100]mm/sec CNT100;
   1:  PR[91,1] = PR[90,1] + 4.385;
   1:  PR[91,2] = PR[90,2] + 7.365;
   1:  PR[91,3] = PR[90,3] + 5.926;
   1:L PR[91] R[100]mm/sec CNT100;
   1:  PR[91,1] = PR[90,1] + 4.060;
   1:  PR[91,2] = PR[90,2] + 6.595;
   1:  PR[91,3] = PR[90,3] + 5.931;
   1:L PR[91] R[100]mm/sec CNT100;
   1:  PR[91,1] = PR[90,1] + 3.773;
   1:  PR[91,2] = PR[90,2] + 5.810;
   1:  PR[91,3] = PR[90,3] + 5.936;
   1:L PR[91] R[100]mm/sec CNT100;
   1:  PR[91,1] = PR[90,1] + 3.526;
   1:  PR[91,2] = PR[90,2] + 5.012;
   1:  PR[91,3] = PR[90,3] + 5.941;
   1:L PR[91] R[100]mm/sec CNT100;
   1:  PR[91,1] = PR[90,1] + 3.318;
   1:  PR[91,2] = PR[90,2] + 4.201;
   1:  PR[91,3] = PR[90,3] + 5.946;
   1:L PR[91] R[100]mm/sec CNT100;
   1:  PR[91,1] = PR[90,1] + 3.065;
   1:  PR[91,2] = PR[90,2] + 3.012;
   1:  PR[91,3] = PR[90,3] + 5.951;
   1:L PR[91] R[100]mm/sec CNT100;
   1:  PR[91,1] = PR[90,1] + 2.921;
   1:  PR[91,2] = PR[90,2] + 2.636;
   1:  PR[91,3] = PR[90,3] + 5.958;
   1:L PR[91] R[100]mm/sec CNT100;
   1:  PR[91,1] = PR[90,1] + 2.733;
   1:  PR[91,2] = PR[90,2] + 2.288;
   1:  PR[91,3] = PR[90,3] + 5.961;
   1:L PR[91] R[100]mm/sec CNT100;
   1:  PR[91,1] = PR[90,1] + 2.500;
   1:  PR[91,2] = PR[90,2] + 1.964;
   1:  PR[91,3] = PR[90,3] + 5.963;
   1:L PR[91] R[100]mm/sec CNT100;
   1:  PR[91,1] = PR[90,1] + 2.236;
   1:  PR[91,2] = PR[90,2] + 1.681;
   1:  PR[91,3] = PR[90,3] + 5.966;
   1:L PR[91] R[100]mm/sec CNT100;
   1:  PR[91,1] = PR[90,1] + 1.934;
   1:  PR[91,2] = PR[90,2] + 1.428;
   1:  PR[91,3] = PR[90,3] + 5.968;
   1:L PR[91] R[100]mm/sec CNT100;
   1:  PR[91,1] = PR[90,1] + 1.601;
   1:  PR[91,2] = PR[90,2] + 1.216;
   1:  PR[91,3] = PR[90,3] + 5.970;
   1:L PR[91] R[100]mm/sec CNT100;
   1:  PR[91,1] = PR[90,1] + 1.245;
   1:  PR[91,2] = PR[90,2] + 1.048;
   1:  PR[91,3] = PR[90,3] + 5.973;
   1:L PR[91] R[100]mm/sec CNT100;
   1:  PR[91,1] = PR[90,1] + 0.870;
   1:  PR[91,2] = PR[90,2] + 0.925;
   1:  PR[91,3] = PR[90,3] + 5.975;
   1:L PR[91] R[100]mm/sec CNT100;
   1:  PR[91,1] = PR[90,1] + 0.483;
   1:  PR[91,2] = PR[90,2] + 0.851;
   1:  PR[91,3] = PR[90,3] + 5.978;
   1:L PR[91] R[100]mm/sec CNT100;
   1:  PR[91,1] = PR[90,1] + 0.109;
   1:  PR[91,2] = PR[90,2] + 0.828;
   1:  PR[91,3] = PR[90,3] + 5.980;
   1:L PR[91] R[100]mm/sec CNT100;
   1:  PR[91,1] = PR[90,1] + -0.348;
   1:  PR[91,3] = PR[90,3] + 5.982;
   1:L PR[91] R[100]mm/sec CNT100;
   1:  PR[91,1] = PR[90,1] + -0.721;
   1:  PR[91,2] = PR[90,2] + 0.851;
   1:  PR[91,3] = PR[90,3] + 5.985;
   1:L PR[91] R[100]mm/sec CNT100;
   1:  PR[91,1] = PR[90,1] + -1.109;
   1:  PR[91,2] = PR[90,2] + 0.925;
   1:  PR[91,3] = PR[90,3] + 5.987;
   1:L PR[91] R[100]mm/sec CNT100;
   1:  PR[91,1] = PR[90,1] + -1.484;
   1:  PR[91,2] = PR[90,2] + 1.048;
   1:  PR[91,3] = PR[90,3] + 5.990;
   1:L PR[91] R[100]mm/sec CNT100;
   1:  PR[91,1] = PR[90,1] + -1.840;
   1:  PR[91,2] = PR[90,2] + 1.216;
   1:  PR[91,3] = PR[90,3] + 5.992;
   1:L PR[91] R[100]mm/sec CNT100;
   1:  PR[91,1] = PR[90,1] + -2.172;
   1:  PR[91,2] = PR[90,2] + 1.428;
   1:  PR[91,3] = PR[90,3] + 5.994;
   1:L PR[91] R[100]mm/sec CNT100;
   1:  PR[91,1] = PR[90,1] + -2.475;
   1:  PR[91,2] = PR[90,2] + 1.681;
   1:  PR[91,3] = PR[90,3] + 5.997;
   1:L PR[91] R[100]mm/sec CNT100;
   1:  PR[91,1] = PR[90,1] + -2.743;
   1:  PR[91,2] = PR[90,2] + 1.969;
   1:  PR[91,3] = PR[90,3] + 5.999;
   1:L PR[91] R[100]mm/sec CNT100;
   1:  PR[91,1] = PR[90,1] + -2.973;
   1:  PR[91,2] = PR[90,2] + 2.290;
   1:  PR[91,3] = PR[90,3] + 6.002;
   1:L PR[91] R[100]mm/sec CNT100;
   1:  PR[91,1] = PR[90,1] + -3.162;
   1:  PR[91,2] = PR[90,2] + 2.641;
   1:  PR[91,3] = PR[90,3] + 6.004;
   1:L PR[91] R[100]mm/sec CNT100;
   1:  PR[91,1] = PR[90,1] + -3.307;
   1:  PR[91,2] = PR[90,2] + 3.024;
   1:  PR[91,3] = PR[90,3] + 6.006;
   1:L PR[91] R[100]mm/sec CNT100;
   1:  PR[91,1] = PR[90,1] + -3.557;
   1:  PR[91,2] = PR[90,2] + 4.201;
   1:  PR[91,3] = PR[90,3] + 6.009;
   1:L PR[91] R[100]mm/sec CNT100;
   1:  PR[91,1] = PR[90,1] + -3.764;
   1:  PR[91,2] = PR[90,2] + 5.012;
   1:  PR[91,3] = PR[90,3] + 6.016;
   1:L PR[91] R[100]mm/sec CNT100;
   1:  PR[91,1] = PR[90,1] + -4.012;
   1:  PR[91,2] = PR[90,2] + 5.810;
   1:  PR[91,3] = PR[90,3] + 6.021;
   1:L PR[91] R[100]mm/sec CNT100;
   1:  PR[91,1] = PR[90,1] + -4.298;
   1:  PR[91,2] = PR[90,2] + 6.595;
   1:  PR[91,3] = PR[90,3] + 6.026;
   1:L PR[91] R[100]mm/sec CNT100;
   1:  PR[91,1] = PR[90,1] + -4.624;
   1:  PR[91,2] = PR[90,2] + 7.365;
   1:  PR[91,3] = PR[90,3] + 6.032;
   1:L PR[91] R[100]mm/sec CNT100;
   1:  PR[91,1] = PR[90,1] + -4.987;
   1:  PR[91,2] = PR[90,2] + 8.119;
   1:  PR[91,3] = PR[90,3] + 6.037;
   1:L PR[91] R[100]mm/sec CNT100;
   1:  PR[91,1] = PR[90,1] + -5.387;
   1:  PR[91,2] = PR[90,2] + 8.855;
   1:  PR[91,3] = PR[90,3] + 6.042;
   1:L PR[91] R[100]mm/sec CNT100;
   1:  PR[91,1] = PR[90,1] + -5.823;
   1:  PR[91,2] = PR[90,2] + 9.569;
   1:  PR[91,3] = PR[90,3] + 6.047;
   1:L PR[91] R[100]mm/sec CNT100;
   1:  PR[91,1] = PR[90,1] + -6.293;
   1:  PR[91,2] = PR[90,2] + 10.261;
   1:  PR[91,3] = PR[90,3] + 6.052;
   1:L PR[91] R[100]mm/sec CNT100;
   1:  PR[91,1] = PR[90,1] + -6.798;
   1:  PR[91,2] = PR[90,2] + 10.930;
   1:  PR[91,3] = PR[90,3] + 6.057;
   1:L PR[91] R[100]mm/sec CNT100;
   1:  PR[91,1] = PR[90,1] + -7.334;
   1:  PR[91,2] = PR[90,2] + 11.572;
   1:  PR[91,3] = PR[90,3] + 6.062;
   1:L PR[91] R[100]mm/sec CNT100;
   1:  PR[91,1] = PR[90,1] + -7.903;
   1:  PR[91,2] = PR[90,2] + 12.187;
   1:  PR[91,3] = PR[90,3] + 6.067;
   1:L PR[91] R[100]mm/sec CNT100;
   1:  PR[91,1] = PR[90,1] + -8.500;
   1:  PR[91,2] = PR[90,2] + 12.772;
   1:  PR[91,3] = PR[90,3] + 6.072;
   1:L PR[91] R[100]mm/sec CNT100;
   1:  PR[91,1] = PR[90,1] + -9.140;
   1:  PR[91,2] = PR[90,2] + 13.339;
   1:  PR[91,3] = PR[90,3] + 6.077;
   1:L PR[91] R[100]mm/sec CNT100;
   1:  PR[91,1] = PR[90,1] + -9.779;
   1:  PR[91,2] = PR[90,2] + 13.853;
   1:  PR[91,3] = PR[90,3] + 6.082;
   1:L PR[91] R[100]mm/sec CNT100;
   1:  PR[91,1] = PR[90,1] + -10.456;
   1:  PR[91,2] = PR[90,2] + 14.344;
   1:  PR[91,3] = PR[90,3] + 6.087;
   1:L PR[91] R[100]mm/sec CNT100;
   1:  PR[91,1] = PR[90,1] + -11.157;
   1:  PR[91,2] = PR[90,2] + 14.802;
   1:  PR[91,3] = PR[90,3] + 6.093;
   1:L PR[91] R[100]mm/sec CNT100;
   1:  PR[91,1] = PR[90,1] + -11.879;
   1:  PR[91,2] = PR[90,2] + 15.224;
   1:  PR[91,3] = PR[90,3] + 6.098;
   1:L PR[91] R[100]mm/sec CNT100;
   1:  PR[91,1] = PR[90,1] + -12.622;
   1:  PR[91,2] = PR[90,2] + 15.610;
   1:  PR[91,3] = PR[90,3] + 6.103;
   1:L PR[91] R[100]mm/sec CNT100;
   1:  PR[91,1] = PR[90,1] + -13.382;
   1:  PR[91,2] = PR[90,2] + 15.960;
   1:  PR[91,3] = PR[90,3] + 6.108;
   1:L PR[91] R[100]mm/sec CNT100;
   1:  PR[91,1] = PR[90,1] + -14.159;
   1:  PR[91,2] = PR[90,2] + 16.271;
   1:  PR[91,3] = PR[90,3] + 6.113;
   1:L PR[91] R[100]mm/sec CNT100;
   1:  PR[91,1] = PR[90,1] + -14.950;
   1:  PR[91,2] = PR[90,2] + 16.543;
   1:  PR[91,3] = PR[90,3] + 6.118;
   1:L PR[91] R[100]mm/sec CNT100;
   1:  PR[91,1] = PR[90,1] + -15.754;
   1:  PR[91,2] = PR[90,2] + 16.776;
   1:  PR[91,3] = PR[90,3] + 6.123;
   1:L PR[91] R[100]mm/sec CNT100;
   1:  PR[91,1] = PR[90,1] + -16.568;
   1:  PR[91,2] = PR[90,2] + 16.969;
   1:  PR[91,3] = PR[90,3] + 6.128;
   1:L PR[91] R[100]mm/sec CNT100;
   1:  PR[91,1] = PR[90,1] + -17.391;
   1:  PR[91,2] = PR[90,2] + 17.122;
   1:  PR[91,3] = PR[90,3] + 6.133;
   1:L PR[91] R[100]mm/sec CNT100;
   1:  PR[91,1] = PR[90,1] + -18.220;
   1:  PR[91,2] = PR[90,2] + 17.234;
   1:  PR[91,3] = PR[90,3] + 6.138;
   1:L PR[91] R[100]mm/sec CNT100;
   1:  PR[91,1] = PR[90,1] + -19.053;
   1:  PR[91,2] = PR[90,2] + 17.305;
   1:  PR[91,3] = PR[90,3] + 6.143;
   1:L PR[91] R[100]mm/sec CNT100;
   1:  PR[91,1] = PR[90,1] + -19.890;
   1:  PR[91,2] = PR[90,2] + 17.334;
   1:  PR[91,3] = PR[90,3] + 6.148;
   1:L PR[91] R[100]mm/sec CNT100;
   1:  PR[91,1] = PR[90,1] + -20.726;
   1:  PR[91,2] = PR[90,2] + 17.322;
   1:  PR[91,3] = PR[90,3] + 6.154;
   1:L PR[91] R[100]mm/sec CNT100;
   1:  PR[91,1] = PR[90,1] + -21.561;
   1:  PR[91,2] = PR[90,2] + 17.269;
   1:  PR[91,3] = PR[90,3] + 6.159;
   1:L PR[91] R[100]mm/sec CNT100;
   1:  PR[91,1] = PR[90,1] + -22.392;
   1:  PR[91,2] = PR[90,2] + 17.175;
   1:  PR[91,3] = PR[90,3] + 6.164;
   1:L PR[91] R[100]mm/sec CNT100;
   1:  PR[91,1] = PR[90,1] + -23.218;
   1:  PR[91,2] = PR[90,2] + 17.040;
   1:  PR[91,3] = PR[90,3] + 6.169;
   1:L PR[91] R[100]mm/sec CNT100;
   1:  PR[91,1] = PR[90,1] + -24.036;
   1:  PR[91,2] = PR[90,2] + 16.865;
   1:  PR[91,3] = PR[90,3] + 6.174;
   1:L PR[91] R[100]mm/sec CNT100;
   1:  PR[91,1] = PR[90,1] + -24.844;
   1:  PR[91,2] = PR[90,2] + 16.649;
   1:  PR[91,3] = PR[90,3] + 6.179;
   1:L PR[91] R[100]mm/sec CNT100;
   1:  PR[91,1] = PR[90,1] + -25.640;
   1:  PR[91,2] = PR[90,2] + 16.393;
   1:  PR[91,3] = PR[90,3] + 6.184;
   1:L PR[91] R[100]mm/sec CNT100;
   1:  PR[91,1] = PR[90,1] + -26.423;
   1:  PR[91,2] = PR[90,2] + 16.099;
   1:  PR[91,3] = PR[90,3] + 6.189;
   1:L PR[91] R[100]mm/sec CNT100;
   1:  PR[91,1] = PR[90,1] + -27.190;
   1:  PR[91,2] = PR[90,2] + 15.766;
   1:  PR[91,3] = PR[90,3] + 6.194;
   1:L PR[91] R[100]mm/sec CNT100;
   1:  PR[91,1] = PR[90,1] + -27.940;
   1:  PR[91,2] = PR[90,2] + 15.396;
   1:  PR[91,3] = PR[90,3] + 6.199;
   1:L PR[91] R[100]mm/sec CNT100;
   1:  PR[91,1] = PR[90,1] + -28.671;
   1:  PR[91,2] = PR[90,2] + 14.990;
   1:  PR[91,3] = PR[90,3] + 6.204;
   1:L PR[91] R[100]mm/sec CNT100;
   1:  PR[91,1] = PR[90,1] + -29.380;
   1:  PR[91,2] = PR[90,2] + 14.547;
   1:  PR[91,3] = PR[90,3] + 6.209;
   1:L PR[91] R[100]mm/sec CNT100;
   1:  PR[91,1] = PR[90,1] + -30.067;
   1:  PR[91,2] = PR[90,2] + 14.071;
   1:  PR[91,3] = PR[90,3] + 6.215;
   1:L PR[91] R[100]mm/sec CNT100;
   1:  PR[91,1] = PR[90,1] + -30.729;
   1:  PR[91,2] = PR[90,2] + 13.561;
   1:  PR[91,3] = PR[90,3] + 6.220;
   1:L PR[91] R[100]mm/sec CNT100;
   1:  PR[91,1] = PR[90,1] + -31.366;
   1:  PR[91,2] = PR[90,2] + 13.019;
   1:  PR[91,3] = PR[90,3] + 6.225;
   1:L PR[91] R[100]mm/sec CNT100;
   1:  PR[91,1] = PR[90,1] + -31.974;
   1:  PR[91,2] = PR[90,2] + 12.446;
   1:  PR[91,3] = PR[90,3] + 6.230;
   1:L PR[91] R[100]mm/sec CNT100;
   1:  PR[91,1] = PR[90,1] + -32.554;
   1:  PR[91,2] = PR[90,2] + 11.844;
   1:  PR[91,3] = PR[90,3] + 6.235;
   1:L PR[91] R[100]mm/sec CNT100;
   1:  PR[91,1] = PR[90,1] + -33.103;
   1:  PR[91,2] = PR[90,2] + 11.214;
   1:  PR[91,3] = PR[90,3] + 6.240;
   1:L PR[91] R[100]mm/sec CNT100;
   1:  PR[91,1] = PR[90,1] + -33.621;
   1:  PR[91,2] = PR[90,2] + 10.557;
   1:  PR[91,3] = PR[90,3] + 6.245;
   1:L PR[91] R[100]mm/sec CNT100;
   1:  PR[91,1] = PR[90,1] + -34.105;
   1:  PR[91,2] = PR[90,2] + 9.876;
   1:  PR[91,3] = PR[90,3] + 6.250;
   1:L PR[91] R[100]mm/sec CNT100;
   1:  PR[91,1] = PR[90,1] + -34.555;
   1:  PR[91,2] = PR[90,2] + 9.172;
   1:  PR[91,3] = PR[90,3] + 6.255;
   1:L PR[91] R[100]mm/sec CNT100;
   1:  PR[91,1] = PR[90,1] + -34.970;
   1:  PR[91,2] = PR[90,2] + 8.446;
   1:  PR[91,3] = PR[90,3] + 6.260;
   1:L PR[91] R[100]mm/sec CNT100;
   1:  PR[91,1] = PR[90,1] + -35.348;
   1:  PR[91,2] = PR[90,2] + 7.701;
   1:  PR[91,3] = PR[90,3] + 6.265;
   1:L PR[91] R[100]mm/sec CNT100;
   1:  PR[91,1] = PR[90,1] + -35.689;
   1:  PR[91,2] = PR[90,2] + 6.939;
   1:  PR[91,3] = PR[90,3] + 6.270;
   1:L PR[91] R[100]mm/sec CNT100;
   1:  PR[91,1] = PR[90,1] + -35.992;
   1:  PR[91,2] = PR[90,2] + 6.160;
   1:  PR[91,3] = PR[90,3] + 6.275;
   1:L PR[91] R[100]mm/sec CNT100;
   1:  PR[91,1] = PR[90,1] + -36.256;
   1:  PR[91,2] = PR[90,2] + 5.367;
   1:  PR[91,3] = PR[90,3] + 6.281;
   1:L PR[91] R[100]mm/sec CNT100;
   1:  PR[91,1] = PR[90,1] + -36.480;
   1:  PR[91,2] = PR[90,2] + 4.564;
   1:  PR[91,3] = PR[90,3] + 6.286;
   1:L PR[91] R[100]mm/sec CNT100;
   1:  PR[91,1] = PR[90,1] + -36.664;
   1:  PR[91,2] = PR[90,2] + 3.749;
   1:  PR[91,3] = PR[90,3] + 6.291;
   1:L PR[91] R[100]mm/sec CNT100;
   1:  PR[91,1] = PR[90,1] + -36.808;
   1:  PR[91,2] = PR[90,2] + 2.927;
   1:  PR[91,3] = PR[90,3] + 6.296;
   1:L PR[91] R[100]mm/sec CNT100;
   1:  PR[91,1] = PR[90,1] + -36.911;
   1:  PR[91,2] = PR[90,2] + 2.098;
   1:  PR[91,3] = PR[90,3] + 6.301;
   1:L PR[91] R[100]mm/sec CNT100;
   1:  PR[91,1] = PR[90,1] + -36.973;
   1:  PR[91,2] = PR[90,2] + 1.264;
   1:  PR[91,3] = PR[90,3] + 6.306;
   1:L PR[91] R[100]mm/sec CNT100;
   1:  PR[91,1] = PR[90,1] + -36.995;
   1:  PR[91,2] = PR[90,2] + 0.428;
   1:  PR[91,3] = PR[90,3] + 6.311;
   1:L PR[91] R[100]mm/sec CNT100;
   1:  PR[91,1] = PR[90,1] + -36.973;
   1:  PR[91,2] = PR[90,2] + -0.409;
   1:  PR[91,3] = PR[90,3] + 6.316;
   1:L PR[91] R[100]mm/sec CNT100;
   1:  PR[91,1] = PR[90,1] + -36.911;
   1:  PR[91,2] = PR[90,2] + -1.242;
   1:  PR[91,3] = PR[90,3] + 6.321;
   1:L PR[91] R[100]mm/sec CNT100;
   1:  PR[91,1] = PR[90,1] + -36.808;
   1:  PR[91,2] = PR[90,2] + -2.072;
   1:  PR[91,3] = PR[90,3] + 6.326;
   1:L PR[91] R[100]mm/sec CNT100;
   1:  PR[91,1] = PR[90,1] + -36.664;
   1:  PR[91,2] = PR[90,2] + -2.894;
   1:  PR[91,3] = PR[90,3] + 6.331;
   1:L PR[91] R[100]mm/sec CNT100;
   1:  PR[91,1] = PR[90,1] + -36.480;
   1:  PR[91,2] = PR[90,2] + -3.708;
   1:  PR[91,3] = PR[90,3] + 6.336;
   1:L PR[91] R[100]mm/sec CNT100;
   1:  PR[91,1] = PR[90,1] + -36.256;
   1:  PR[91,2] = PR[90,2] + -4.512;
   1:  PR[91,3] = PR[90,3] + 6.341;
   1:L PR[91] R[100]mm/sec CNT100;
   1:  PR[91,1] = PR[90,1] + -35.992;
   1:  PR[91,2] = PR[90,2] + -5.305;
   1:  PR[91,3] = PR[90,3] + 6.347;
   1:L PR[91] R[100]mm/sec CNT100;
   1:  PR[91,1] = PR[90,1] + -35.689;
   1:  PR[91,2] = PR[90,2] + -6.083;
   1:  PR[91,3] = PR[90,3] + 6.352;
   1:L PR[91] R[100]mm/sec CNT100;
   1:  PR[91,1] = PR[90,1] + -35.348;
   1:  PR[91,2] = PR[90,2] + -6.846;
   1:  PR[91,3] = PR[90,3] + 6.357;
   1:L PR[91] R[100]mm/sec CNT100;
   1:  PR[91,1] = PR[90,1] + -34.970;
   1:  PR[91,2] = PR[90,2] + -7.591;
   1:  PR[91,3] = PR[90,3] + 6.362;
   1:L PR[91] R[100]mm/sec CNT100;
   1:  PR[91,1] = PR[90,1] + -34.555;
   1:  PR[91,2] = PR[90,2] + -8.317;
   1:  PR[91,3] = PR[90,3] + 6.367;
   1:L PR[91] R[100]mm/sec CNT100;
   1:  PR[91,1] = PR[90,1] + -34.105;
   1:  PR[91,2] = PR[90,2] + -9.021;
   1:  PR[91,3] = PR[90,3] + 6.372;
   1:L PR[91] R[100]mm/sec CNT100;
   1:  PR[91,1] = PR[90,1] + -33.621;
   1:  PR[91,2] = PR[90,2] + -9.702;
   1:  PR[91,3] = PR[90,3] + 6.377;
   1:L PR[91] R[100]mm/sec CNT100;
   1:  PR[91,1] = PR[90,1] + -33.103;
   1:  PR[91,2] = PR[90,2] + -10.359;
   1:  PR[91,3] = PR[90,3] + 6.382;
   1:L PR[91] R[100]mm/sec CNT100;
   1:  PR[91,1] = PR[90,1] + -32.554;
   1:  PR[91,2] = PR[90,2] + -10.989;
   1:  PR[91,3] = PR[90,3] + 6.387;
   1:L PR[91] R[100]mm/sec CNT100;
   1:  PR[91,1] = PR[90,1] + -31.974;
   1:  PR[91,2] = PR[90,2] + -11.591;
   1:  PR[91,3] = PR[90,3] + 6.392;
   1:L PR[91] R[100]mm/sec CNT100;
   1:  PR[91,1] = PR[90,1] + -31.366;
   1:  PR[91,2] = PR[90,2] + -12.164;
   1:  PR[91,3] = PR[90,3] + 6.397;
   1:L PR[91] R[100]mm/sec CNT100;
   1:  PR[91,1] = PR[90,1] + -30.729;
   1:  PR[91,2] = PR[90,2] + -12.706;
   1:  PR[91,3] = PR[90,3] + 6.402;
   1:L PR[91] R[100]mm/sec CNT100;
   1:  PR[91,1] = PR[90,1] + -30.067;
   1:  PR[91,2] = PR[90,2] + -13.216;
   1:  PR[91,3] = PR[90,3] + 6.408;
   1:L PR[91] R[100]mm/sec CNT100;
   1:  PR[91,1] = PR[90,1] + -29.380;
   1:  PR[91,2] = PR[90,2] + -13.692;
   1:  PR[91,3] = PR[90,3] + 6.413;
   1:L PR[91] R[100]mm/sec CNT100;
   1:  PR[91,1] = PR[90,1] + -28.671;
   1:  PR[91,2] = PR[90,2] + -14.134;
   1:  PR[91,3] = PR[90,3] + 6.418;
   1:L PR[91] R[100]mm/sec CNT100;
   1:  PR[91,1] = PR[90,1] + -27.940;
   1:  PR[91,2] = PR[90,2] + -14.541;
   1:  PR[91,3] = PR[90,3] + 6.423;
   1:L PR[91] R[100]mm/sec CNT100;
   1:  PR[91,1] = PR[90,1] + -27.190;
   1:  PR[91,2] = PR[90,2] + -14.911;
   1:  PR[91,3] = PR[90,3] + 6.428;
   1:L PR[91] R[100]mm/sec CNT100;
   1:  PR[91,1] = PR[90,1] + -26.423;
   1:  PR[91,2] = PR[90,2] + -15.244;
   1:  PR[91,3] = PR[90,3] + 6.433;
   1:L PR[91] R[100]mm/sec CNT100;
   1:  PR[91,1] = PR[90,1] + -25.640;
   1:  PR[91,2] = PR[90,2] + -15.538;
   1:  PR[91,3] = PR[90,3] + 6.438;
   1:L PR[91] R[100]mm/sec CNT100;
   1:  PR[91,1] = PR[90,1] + -24.844;
   1:  PR[91,2] = PR[90,2] + -15.794;
   1:  PR[91,3] = PR[90,3] + 6.443;
   1:L PR[91] R[100]mm/sec CNT100;
   1:  PR[91,1] = PR[90,1] + -24.036;
   1:  PR[91,2] = PR[90,2] + -16.009;
   1:  PR[91,3] = PR[90,3] + 6.448;
   1:L PR[91] R[100]mm/sec CNT100;
   1:  PR[91,1] = PR[90,1] + -23.218;
   1:  PR[91,2] = PR[90,2] + -16.185;
   1:  PR[91,3] = PR[90,3] + 6.453;
   1:L PR[91] R[100]mm/sec CNT100;
   1:  PR[91,1] = PR[90,1] + -22.392;
   1:  PR[91,2] = PR[90,2] + -16.320;
   1:  PR[91,3] = PR[90,3] + 6.458;
   1:L PR[91] R[100]mm/sec CNT100;
   1:  PR[91,1] = PR[90,1] + -21.561;
   1:  PR[91,2] = PR[90,2] + -16.414;
   1:  PR[91,3] = PR[90,3] + 6.463;
   1:L PR[91] R[100]mm/sec CNT100;
   1:  PR[91,1] = PR[90,1] + -20.726;
   1:  PR[91,2] = PR[90,2] + -16.467;
   1:  PR[91,3] = PR[90,3] + 6.468;
   1:L PR[91] R[100]mm/sec CNT100;
   1:  PR[91,1] = PR[90,1] + -19.890;
   1:  PR[91,2] = PR[90,2] + -16.479;
   1:  PR[91,3] = PR[90,3] + 6.474;
   1:L PR[91] R[100]mm/sec CNT100;
   1:  PR[91,1] = PR[90,1] + -19.054;
   1:  PR[91,2] = PR[90,2] + -16.449;
   1:  PR[91,3] = PR[90,3] + 6.479;
   1:L PR[91] R[100]mm/sec CNT100;
   1:  PR[91,1] = PR[90,1] + -18.220;
   1:  PR[91,2] = PR[90,2] + -16.379;
   1:  PR[91,3] = PR[90,3] + 6.484;
   1:L PR[91] R[100]mm/sec CNT100;
   1:  PR[91,1] = PR[90,1] + -17.391;
   1:  PR[91,2] = PR[90,2] + -16.267;
   1:  PR[91,3] = PR[90,3] + 6.489;
   1:L PR[91] R[100]mm/sec CNT100;
   1:  PR[91,1] = PR[90,1] + -16.568;
   1:  PR[91,2] = PR[90,2] + -16.114;
   1:  PR[91,3] = PR[90,3] + 6.494;
   1:L PR[91] R[100]mm/sec CNT100;
   1:  PR[91,1] = PR[90,1] + -15.754;
   1:  PR[91,2] = PR[90,2] + -15.921;
   1:  PR[91,3] = PR[90,3] + 6.499;
   1:L PR[91] R[100]mm/sec CNT100;
   1:  PR[91,1] = PR[90,1] + -14.950;
   1:  PR[91,2] = PR[90,2] + -15.688;
   1:  PR[91,3] = PR[90,3] + 6.504;
   1:L PR[91] R[100]mm/sec CNT100;
   1:  PR[91,1] = PR[90,1] + -14.159;
   1:  PR[91,2] = PR[90,2] + -15.416;
   1:  PR[91,3] = PR[90,3] + 6.509;
   1:L PR[91] R[100]mm/sec CNT100;
   1:  PR[91,1] = PR[90,1] + -13.382;
   1:  PR[91,2] = PR[90,2] + -15.105;
   1:  PR[91,3] = PR[90,3] + 6.514;
   1:L PR[91] R[100]mm/sec CNT100;
   1:  PR[91,1] = PR[90,1] + -12.622;
   1:  PR[91,2] = PR[90,2] + -14.755;
   1:  PR[91,3] = PR[90,3] + 6.519;
   1:L PR[91] R[100]mm/sec CNT100;
   1:  PR[91,1] = PR[90,1] + -11.879;
   1:  PR[91,2] = PR[90,2] + -14.369;
   1:  PR[91,3] = PR[90,3] + 6.524;
   1:L PR[91] R[100]mm/sec CNT100;
   1:  PR[91,1] = PR[90,1] + -11.157;
   1:  PR[91,2] = PR[90,2] + -13.947;
   1:  PR[91,3] = PR[90,3] + 6.530;
   1:L PR[91] R[100]mm/sec CNT100;
   1:  PR[91,1] = PR[90,1] + -10.456;
   1:  PR[91,2] = PR[90,2] + -13.489;
   1:  PR[91,3] = PR[90,3] + 6.535;
   1:L PR[91] R[100]mm/sec CNT100;
   1:  PR[91,1] = PR[90,1] + -9.778;
   1:  PR[91,2] = PR[90,2] + -12.997;
   1:  PR[91,3] = PR[90,3] + 6.540;
   1:L PR[91] R[100]mm/sec CNT100;
   1:  PR[91,1] = PR[90,1] + -9.126;
   1:  PR[91,2] = PR[90,2] + -12.473;
   1:  PR[91,3] = PR[90,3] + 6.545;
   1:L PR[91] R[100]mm/sec CNT100;
   1:  PR[91,1] = PR[90,1] + -8.500;
   1:  PR[91,2] = PR[90,2] + -11.918;
   1:  PR[91,3] = PR[90,3] + 6.550;
   1:L PR[91] R[100]mm/sec CNT100;
   1:  PR[91,1] = PR[90,1] + -7.903;
   1:  PR[91,2] = PR[90,2] + -11.332;
   1:  PR[91,3] = PR[90,3] + 6.555;
   1:L PR[91] R[100]mm/sec CNT100;
   1:  PR[91,1] = PR[90,1] + -7.334;
   1:  PR[91,2] = PR[90,2] + -10.717;
   1:  PR[91,3] = PR[90,3] + 6.560;
   1:L PR[91] R[100]mm/sec CNT100;
   1:  PR[91,1] = PR[90,1] + -6.798;
   1:  PR[91,2] = PR[90,2] + -10.074;
   1:  PR[91,3] = PR[90,3] + 6.565;
   1:L PR[91] R[100]mm/sec CNT100;
   1:  PR[91,1] = PR[90,1] + -6.293;
   1:  PR[91,2] = PR[90,2] + -9.406;
   1:  PR[91,3] = PR[90,3] + 6.570;
   1:L PR[91] R[100]mm/sec CNT100;
   1:  PR[91,1] = PR[90,1] + -5.823;
   1:  PR[91,2] = PR[90,2] + -8.714;
   1:  PR[91,3] = PR[90,3] + 6.575;
   1:L PR[91] R[100]mm/sec CNT100;
   1:  PR[91,1] = PR[90,1] + -5.387;
   1:  PR[91,2] = PR[90,2] + -8.000;
   1:  PR[91,3] = PR[90,3] + 6.580;
   1:L PR[91] R[100]mm/sec CNT100;
   1:  PR[91,1] = PR[90,1] + -4.987;
   1:  PR[91,2] = PR[90,2] + -7.264;
   1:  PR[91,3] = PR[90,3] + 6.585;
   1:L PR[91] R[100]mm/sec CNT100;
   1:  PR[91,1] = PR[90,1] + -4.624;
   1:  PR[91,2] = PR[90,2] + -6.510;
   1:  PR[91,3] = PR[90,3] + 6.591;
   1:L PR[91] R[100]mm/sec CNT100;
   1:  PR[91,1] = PR[90,1] + -4.298;
   1:  PR[91,2] = PR[90,2] + -5.740;
   1:  PR[91,3] = PR[90,3] + 6.596;
   1:L PR[91] R[100]mm/sec CNT100;
   1:  PR[91,1] = PR[90,1] + -4.012;
   1:  PR[91,2] = PR[90,2] + -4.955;
   1:  PR[91,3] = PR[90,3] + 6.601;
   1:L PR[91] R[100]mm/sec CNT100;
   1:  PR[91,1] = PR[90,1] + -3.764;
   1:  PR[91,2] = PR[90,2] + -4.157;
   1:  PR[91,3] = PR[90,3] + 6.606;
   1:L PR[91] R[100]mm/sec CNT100;
   1:  PR[91,1] = PR[90,1] + -3.557;
   1:  PR[91,2] = PR[90,2] + -3.345;
   1:  PR[91,3] = PR[90,3] + 6.611;
   1:L PR[91] R[100]mm/sec CNT100;
   1:  PR[91,1] = PR[90,1] + -3.304;
   1:  PR[91,2] = PR[90,2] + -2.157;
   1:  PR[91,3] = PR[90,3] + 6.616;
   1:L PR[91] R[100]mm/sec CNT100;
   1:  PR[91,1] = PR[90,1] + -3.160;
   1:  PR[91,2] = PR[90,2] + -1.781;
   1:  PR[91,3] = PR[90,3] + 6.623;
   1:L PR[91] R[100]mm/sec CNT100;
   1:  PR[91,1] = PR[90,1] + -2.972;
   1:  PR[91,2] = PR[90,2] + -1.432;
   1:  PR[91,3] = PR[90,3] + 6.626;
   1:L PR[91] R[100]mm/sec CNT100;
   1:  PR[91,1] = PR[90,1] + -2.738;
   1:  PR[91,2] = PR[90,2] + -1.108;
   1:  PR[91,3] = PR[90,3] + 6.628;
   1:L PR[91] R[100]mm/sec CNT100;
   1:  PR[91,1] = PR[90,1] + -2.475;
   1:  PR[91,2] = PR[90,2] + -0.825;
   1:  PR[91,3] = PR[90,3] + 6.631;
   1:L PR[91] R[100]mm/sec CNT100;
   1:  PR[91,1] = PR[90,1] + -2.172;
   1:  PR[91,2] = PR[90,2] + -0.573;
   1:  PR[91,3] = PR[90,3] + 6.633;
   1:L PR[91] R[100]mm/sec CNT100;
   1:  PR[91,1] = PR[90,1] + -1.840;
   1:  PR[91,2] = PR[90,2] + -0.361;
   1:  PR[91,3] = PR[90,3] + 6.635;
   1:L PR[91] R[100]mm/sec CNT100;
   1:  PR[91,1] = PR[90,1] + -1.484;
   1:  PR[91,2] = PR[90,2] + -0.193;
   1:  PR[91,3] = PR[90,3] + 6.638;
   1:L PR[91] R[100]mm/sec CNT100;
   1:  PR[91,1] = PR[90,1] + -1.109;
   1:  PR[91,2] = PR[90,2] + -0.070;
   1:  PR[91,3] = PR[90,3] + 6.640;
   1:L PR[91] R[100]mm/sec CNT100;
   1:  PR[91,1] = PR[90,1] + -0.721;
   1:  PR[91,2] = PR[90,2] + 0.004;
   1:  PR[91,3] = PR[90,3] + 6.643;
   1:L PR[91] R[100]mm/sec CNT100;
   1:  PR[91,1] = PR[90,1] + -0.348;
   1:  PR[91,2] = PR[90,2] + 0.028;
   1:  PR[91,3] = PR[90,3] + 6.645;
   1:L PR[91] R[100]mm/sec CNT100;
   1:  PR[91,1] = PR[90,1] + 0.109;
   1:  PR[91,3] = PR[90,3] + 6.647;
   1:L PR[91] R[100]mm/sec CNT100;
   1:  PR[91] = PR[90];
   1:  PR[91,1] = PR[90,1] + 0.713;
   1:  PR[91,2] = PR[90,2] + -0.072;
   1:  PR[91,3] = PR[90,3] + 7.980;
   1:L PR[91] R[100]mm/sec CNT100;
   1:  PR[91,1] = PR[90,1] + 0.941;
   1:  PR[91,2] = PR[90,2] + -0.144;
   1:  PR[91,3] = PR[90,3] + 6.653;
   1:L PR[91] R[100]mm/sec CNT100;
   1:  PR[91,1] = PR[90,1] + 1.166;
   1:  PR[91,2] = PR[90,2] + -0.229;
   1:  PR[91,3] = PR[90,3] + 6.654;
   1:L PR[91] R[100]mm/sec CNT100;
   1:  PR[91,1] = PR[90,1] + 1.463;
   1:  PR[91,2] = PR[90,2] + -0.374;
   1:  PR[91,3] = PR[90,3] + 6.656;
   1:L PR[91] R[100]mm/sec CNT100;
   1:  PR[91,1] = PR[90,1] + 1.802;
   1:  PR[91,2] = PR[90,2] + -0.595;
   1:  PR[91,3] = PR[90,3] + 6.658;
   1:L PR[91] R[100]mm/sec CNT100;
   1:  PR[91,1] = PR[90,1] + 2.097;
   1:  PR[91,2] = PR[90,2] + -0.845;
   1:  PR[91,3] = PR[90,3] + 6.660;
   1:L PR[91] R[100]mm/sec CNT100;
   1:  PR[91,1] = PR[90,1] + 2.336;
   1:  PR[91,2] = PR[90,2] + -1.102;
   1:  PR[91,3] = PR[90,3] + 6.662;
   1:L PR[91] R[100]mm/sec CNT100;
   1:  PR[91,1] = PR[90,1] + 2.583;
   1:  PR[91,2] = PR[90,2] + -1.444;
   1:  PR[91,3] = PR[90,3] + 6.665;
   1:L PR[91] R[100]mm/sec CNT100;
   1:  PR[91,1] = PR[90,1] + 2.763;
   1:  PR[91,2] = PR[90,2] + -1.777;
   1:  PR[91,3] = PR[90,3] + 6.667;
   1:L PR[91] R[100]mm/sec CNT100;
   1:  PR[91,1] = PR[90,1] + 2.919;
   1:  PR[91,2] = PR[90,2] + -2.189;
   1:  PR[91,3] = PR[90,3] + 6.669;
   1:L PR[91] R[100]mm/sec CNT100;
   1:  PR[91,1] = PR[90,1] + 3.168;
   1:  PR[91,2] = PR[90,2] + -3.346;
   1:  PR[91,3] = PR[90,3] + 6.672;
   1:L PR[91] R[100]mm/sec CNT100;
   1:  PR[91,1] = PR[90,1] + 3.376;
   1:  PR[91,2] = PR[90,2] + -4.157;
   1:  PR[91,3] = PR[90,3] + 6.679;
   1:L PR[91] R[100]mm/sec CNT100;
   1:  PR[91,1] = PR[90,1] + 3.625;
   1:  PR[91,2] = PR[90,2] + -4.954;
   1:  PR[91,3] = PR[90,3] + 6.684;
   1:L PR[91] R[100]mm/sec CNT100;
   1:  PR[91,1] = PR[90,1] + 3.913;
   1:  PR[91,2] = PR[90,2] + -5.739;
   1:  PR[91,3] = PR[90,3] + 6.689;
   1:L PR[91] R[100]mm/sec CNT100;
   1:  PR[91,1] = PR[90,1] + 4.240;
   1:  PR[91,2] = PR[90,2] + -6.510;
   1:  PR[91,3] = PR[90,3] + 6.695;
   1:L PR[91] R[100]mm/sec CNT100;
   1:  PR[91,1] = PR[90,1] + 4.604;
   1:  PR[91,2] = PR[90,2] + -7.265;
   1:  PR[91,3] = PR[90,3] + 6.700;
   1:L PR[91] R[100]mm/sec CNT100;
   1:  PR[91,1] = PR[90,1] + 5.007;
   1:  PR[91,2] = PR[90,2] + -8.002;
   1:  PR[91,3] = PR[90,3] + 6.705;
   1:L PR[91] R[100]mm/sec CNT100;
   1:  PR[91,1] = PR[90,1] + 5.445;
   1:  PR[91,2] = PR[90,2] + -8.718;
   1:  PR[91,3] = PR[90,3] + 6.710;
   1:L PR[91] R[100]mm/sec CNT100;
   1:  PR[91,1] = PR[90,1] + 5.918;
   1:  PR[91,2] = PR[90,2] + -9.413;
   1:  PR[91,3] = PR[90,3] + 6.715;
   1:L PR[91] R[100]mm/sec CNT100;
   1:  PR[91,1] = PR[90,1] + 6.425;
   1:  PR[91,2] = PR[90,2] + -10.082;
   1:  PR[91,3] = PR[90,3] + 6.720;
   1:L PR[91] R[100]mm/sec CNT100;
   1:  PR[91,1] = PR[90,1] + 6.965;
   1:  PR[91,2] = PR[90,2] + -10.726;
   1:  PR[91,3] = PR[90,3] + 6.725;
   1:L PR[91] R[100]mm/sec CNT100;
   1:  PR[91,1] = PR[90,1] + 7.535;
   1:  PR[91,2] = PR[90,2] + -11.343;
   1:  PR[91,3] = PR[90,3] + 6.730;
   1:L PR[91] R[100]mm/sec CNT100;
   1:  PR[91,1] = PR[90,1] + 8.136;
   1:  PR[91,2] = PR[90,2] + -11.930;
   1:  PR[91,3] = PR[90,3] + 6.735;
   1:L PR[91] R[100]mm/sec CNT100;
   1:  PR[91,1] = PR[90,1] + 8.765;
   1:  PR[91,2] = PR[90,2] + -12.486;
   1:  PR[91,3] = PR[90,3] + 6.740;
   1:L PR[91] R[100]mm/sec CNT100;
   1:  PR[91,1] = PR[90,1] + 9.421;
   1:  PR[91,2] = PR[90,2] + -13.011;
   1:  PR[91,3] = PR[90,3] + 6.746;
   1:L PR[91] R[100]mm/sec CNT100;
   1:  PR[91,1] = PR[90,1] + 10.102;
   1:  PR[91,2] = PR[90,2] + -13.503;
   1:  PR[91,3] = PR[90,3] + 6.751;
   1:L PR[91] R[100]mm/sec CNT100;
   1:  PR[91,1] = PR[90,1] + 10.807;
   1:  PR[91,2] = PR[90,2] + -13.961;
   1:  PR[91,3] = PR[90,3] + 6.756;
   1:L PR[91] R[100]mm/sec CNT100;
   1:  PR[91,1] = PR[90,1] + 11.533;
   1:  PR[91,2] = PR[90,2] + -14.383;
   1:  PR[91,3] = PR[90,3] + 6.761;
   1:L PR[91] R[100]mm/sec CNT100;
   1:  PR[91,1] = PR[90,1] + 12.280;
   1:  PR[91,2] = PR[90,2] + -14.769;
   1:  PR[91,3] = PR[90,3] + 6.766;
   1:L PR[91] R[100]mm/sec CNT100;
   1:  PR[91,1] = PR[90,1] + 13.044;
   1:  PR[91,2] = PR[90,2] + -15.119;
   1:  PR[91,3] = PR[90,3] + 6.771;
   1:L PR[91] R[100]mm/sec CNT100;
   1:  PR[91,1] = PR[90,1] + 13.825;
   1:  PR[91,2] = PR[90,2] + -15.430;
   1:  PR[91,3] = PR[90,3] + 6.776;
   1:L PR[91] R[100]mm/sec CNT100;
   1:  PR[91,1] = PR[90,1] + 14.620;
   1:  PR[91,2] = PR[90,2] + -15.702;
   1:  PR[91,3] = PR[90,3] + 6.781;
   1:L PR[91] R[100]mm/sec CNT100;
   1:  PR[91,1] = PR[90,1] + 15.440;
   1:  PR[91,2] = PR[90,2] + -15.938;
   1:  PR[91,3] = PR[90,3] + 6.786;
   1:L PR[91] R[100]mm/sec CNT100;
   1:  PR[91,1] = PR[90,1] + 16.245;
   1:  PR[91,2] = PR[90,2] + -16.128;
   1:  PR[91,3] = PR[90,3] + 6.792;
   1:L PR[91] R[100]mm/sec CNT100;
   1:  PR[91,1] = PR[90,1] + 17.071;
   1:  PR[91,2] = PR[90,2] + -16.280;
   1:  PR[91,3] = PR[90,3] + 6.797;
   1:L PR[91] R[100]mm/sec CNT100;
   1:  PR[91,1] = PR[90,1] + 17.903;
   1:  PR[91,2] = PR[90,2] + -16.392;
   1:  PR[91,3] = PR[90,3] + 6.802;
   1:L PR[91] R[100]mm/sec CNT100;
   1:  PR[91,1] = PR[90,1] + 18.739;
   1:  PR[91,2] = PR[90,2] + -16.463;
   1:  PR[91,3] = PR[90,3] + 6.807;
   1:L PR[91] R[100]mm/sec CNT100;
   1:  PR[91,1] = PR[90,1] + 19.577;
   1:  PR[91,2] = PR[90,2] + -16.492;
   1:  PR[91,3] = PR[90,3] + 6.812;
   1:L PR[91] R[100]mm/sec CNT100;
   1:  PR[91,1] = PR[90,1] + 20.416;
   1:  PR[91,2] = PR[90,2] + -16.480;
   1:  PR[91,3] = PR[90,3] + 6.817;
   1:L PR[91] R[100]mm/sec CNT100;
   1:  PR[91,1] = PR[90,1] + 21.253;
   1:  PR[91,2] = PR[90,2] + -16.426;
   1:  PR[91,3] = PR[90,3] + 6.822;
   1:L PR[91] R[100]mm/sec CNT100;
   1:  PR[91,1] = PR[90,1] + 22.086;
   1:  PR[91,2] = PR[90,2] + -16.332;
   1:  PR[91,3] = PR[90,3] + 6.827;
   1:L PR[91] R[100]mm/sec CNT100;
   1:  PR[91,1] = PR[90,1] + 22.914;
   1:  PR[91,2] = PR[90,2] + -16.196;
   1:  PR[91,3] = PR[90,3] + 6.832;
   1:L PR[91] R[100]mm/sec CNT100;
   1:  PR[91,1] = PR[90,1] + 23.734;
   1:  PR[91,2] = PR[90,2] + -16.020;
   1:  PR[91,3] = PR[90,3] + 6.838;
   1:L PR[91] R[100]mm/sec CNT100;
   1:  PR[91,1] = PR[90,1] + 24.544;
   1:  PR[91,2] = PR[90,2] + -15.804;
   1:  PR[91,3] = PR[90,3] + 6.843;
   1:L PR[91] R[100]mm/sec CNT100;
   1:  PR[91,1] = PR[90,1] + 25.342;
   1:  PR[91,2] = PR[90,2] + -15.548;
   1:  PR[91,3] = PR[90,3] + 6.848;
   1:L PR[91] R[100]mm/sec CNT100;
   1:  PR[91,1] = PR[90,1] + 26.126;
   1:  PR[91,2] = PR[90,2] + -15.253;
   1:  PR[91,3] = PR[90,3] + 6.853;
   1:L PR[91] R[100]mm/sec CNT100;
   1:  PR[91,1] = PR[90,1] + 26.895;
   1:  PR[91,2] = PR[90,2] + -14.920;
   1:  PR[91,3] = PR[90,3] + 6.858;
   1:L PR[91] R[100]mm/sec CNT100;
   1:  PR[91,1] = PR[90,1] + 27.647;
   1:  PR[91,2] = PR[90,2] + -14.549;
   1:  PR[91,3] = PR[90,3] + 6.863;
   1:L PR[91] R[100]mm/sec CNT100;
   1:  PR[91,1] = PR[90,1] + 28.379;
   1:  PR[91,2] = PR[90,2] + -14.142;
   1:  PR[91,3] = PR[90,3] + 6.868;
   1:L PR[91] R[100]mm/sec CNT100;
   1:  PR[91,1] = PR[90,1] + 29.090;
   1:  PR[91,2] = PR[90,2] + -13.700;
   1:  PR[91,3] = PR[90,3] + 6.873;
   1:L PR[91] R[100]mm/sec CNT100;
   1:  PR[91,1] = PR[90,1] + 29.778;
   1:  PR[91,2] = PR[90,2] + -13.223;
   1:  PR[91,3] = PR[90,3] + 6.878;
   1:L PR[91] R[100]mm/sec CNT100;
   1:  PR[91,1] = PR[90,1] + 30.441;
   1:  PR[91,2] = PR[90,2] + -12.712;
   1:  PR[91,3] = PR[90,3] + 6.883;
   1:L PR[91] R[100]mm/sec CNT100;
   1:  PR[91,1] = PR[90,1] + 31.079;
   1:  PR[91,2] = PR[90,2] + -12.170;
   1:  PR[91,3] = PR[90,3] + 6.888;
   1:L PR[91] R[100]mm/sec CNT100;
   1:  PR[91,1] = PR[90,1] + 31.689;
   1:  PR[91,2] = PR[90,2] + -11.597;
   1:  PR[91,3] = PR[90,3] + 6.894;
   1:L PR[91] R[100]mm/sec CNT100;
   1:  PR[91,1] = PR[90,1] + 32.269;
   1:  PR[91,2] = PR[90,2] + -10.994;
   1:  PR[91,3] = PR[90,3] + 6.899;
   1:L PR[91] R[100]mm/sec CNT100;
   1:  PR[91,1] = PR[90,1] + 32.819;
   1:  PR[91,2] = PR[90,2] + -10.363;
   1:  PR[91,3] = PR[90,3] + 6.904;
   1:L PR[91] R[100]mm/sec CNT100;
   1:  PR[91,1] = PR[90,1] + 33.337;
   1:  PR[91,2] = PR[90,2] + -9.706;
   1:  PR[91,3] = PR[90,3] + 6.909;
   1:L PR[91] R[100]mm/sec CNT100;
   1:  PR[91,1] = PR[90,1] + 33.822;
   1:  PR[91,2] = PR[90,2] + -9.024;
   1:  PR[91,3] = PR[90,3] + 6.914;
   1:L PR[91] R[100]mm/sec CNT100;
   1:  PR[91,1] = PR[90,1] + 34.273;
